LIN {X 272.582,Y -98.990,Z 143.292,A 160.041,B 90.000,C 0.000} C_DIS
LIN {X 272.604,Y -98.930,Z 143.343,A 160.054,B 90.000,C 0.000} C_DIS
LIN {X 272.618,Y -98.890,Z 143.394,A 160.062,B 90.000,C 0.000} C_DIS
LIN {X 272.688,Y -98.698,Z 143.436,A 160.103,B 90.000,C 0.000} C_DIS
LIN {X 272.717,Y -98.618,Z 143.538,A 160.119,B 90.000,C 0.000} C_DIS
LIN {X 272.786,Y -98.426,Z 143.581,A 160.160,B 90.000,C 0.000} C_DIS
LIN {X 272.801,Y -98.386,Z 143.632,A 160.168,B 90.000,C 0.000} C_DIS
LIN {X 272.822,Y -98.326,Z 143.683,A 160.181,B 90.000,C 0.000} C_DIS
LIN {X 272.926,Y -98.038,Z 143.725,A 160.241,B 90.000,C 0.000} C_DIS
LIN {X 272.947,Y -97.978,Z 143.776,A 160.254,B 90.000,C 0.000} C_DIS
LIN {X 272.962,Y -97.938,Z 143.827,A 160.262,B 90.000,C 0.000} C_DIS
LIN {X 273.031,Y -97.746,Z 143.870,A 160.302,B 90.000,C 0.000} C_DIS
LIN {X 273.059,Y -97.666,Z 143.972,A 160.319,B 90.000,C 0.000} C_DIS
LIN {X 273.128,Y -97.474,Z 144.014,A 160.360,B 90.000,C 0.000} C_DIS
LIN {X 273.142,Y -97.434,Z 144.065,A 160.368,B 90.000,C 0.000} C_DIS
LIN {X 273.164,Y -97.374,Z 144.116,A 160.380,B 90.000,C 0.000} C_DIS
LIN {X 273.266,Y -97.086,Z 144.159,A 160.441,B 90.000,C 0.000} C_DIS
LIN {X 273.287,Y -97.026,Z 144.210,A 160.454,B 90.000,C 0.000} C_DIS
LIN {X 273.302,Y -96.986,Z 144.261,A 160.462,B 90.000,C 0.000} C_DIS
LIN {X 273.370,Y -96.793,Z 144.303,A 160.502,B 90.000,C 0.000} C_DIS
LIN {X 273.398,Y -96.713,Z 144.405,A 160.519,B 90.000,C 0.000} C_DIS
LIN {X 273.466,Y -96.521,Z 144.448,A 160.559,B 90.000,C 0.000} C_DIS
LIN {X 273.480,Y -96.481,Z 144.499,A 160.568,B 90.000,C 0.000} C_DIS
LIN {X 273.502,Y -96.420,Z 144.550,A 160.580,B 90.000,C 0.000} C_DIS
LIN {X 273.603,Y -96.132,Z 144.592,A 160.641,B 90.000,C 0.000} C_DIS
LIN {X 273.624,Y -96.072,Z 144.644,A 160.653,B 90.000,C 0.000} C_DIS
LIN {X 273.638,Y -96.031,Z 144.695,A 160.662,B 90.000,C 0.000} C_DIS
LIN {X 273.706,Y -95.839,Z 144.737,A 160.702,B 90.000,C 0.000} C_DIS
LIN {X 273.734,Y -95.759,Z 144.839,A 160.719,B 90.000,C 0.000} C_DIS
LIN {X 273.801,Y -95.566,Z 144.882,A 160.759,B 90.000,C 0.000} C_DIS
LIN {X 273.815,Y -95.526,Z 144.933,A 160.768,B 90.000,C 0.000} C_DIS
LIN {X 273.836,Y -95.466,Z 144.984,A 160.780,B 90.000,C 0.000} C_DIS
LIN {X 273.937,Y -95.177,Z 145.026,A 160.841,B 90.000,C 0.000} C_DIS
LIN {X 273.958,Y -95.116,Z 145.077,A 160.853,B 90.000,C 0.000} C_DIS
LIN {X 273.972,Y -95.076,Z 145.128,A 160.862,B 90.000,C 0.000} C_DIS
LIN {X 274.039,Y -94.883,Z 145.171,A 160.902,B 90.000,C 0.000} C_DIS
LIN {X 274.066,Y -94.803,Z 145.273,A 160.919,B 90.000,C 0.000} C_DIS
LIN {X 274.133,Y -94.610,Z 145.315,A 160.959,B 90.000,C 0.000} C_DIS
LIN {X 274.161,Y -94.530,Z 145.417,A 160.976,B 90.000,C 0.000} C_DIS
LIN {X 274.227,Y -94.337,Z 145.460,A 161.016,B 90.000,C 0.000} C_DIS
LIN {X 274.241,Y -94.297,Z 145.511,A 161.025,B 90.000,C 0.000} C_DIS
LIN {X 274.262,Y -94.237,Z 145.562,A 161.037,B 90.000,C 0.000} C_DIS
LIN {X 274.361,Y -93.947,Z 145.604,A 161.098,B 90.000,C 0.000} C_DIS
LIN {X 274.382,Y -93.887,Z 145.655,A 161.110,B 90.000,C 0.000} C_DIS
LIN {X 274.395,Y -93.846,Z 145.706,A 161.119,B 90.000,C 0.000} C_DIS
LIN {X 274.461,Y -93.653,Z 145.749,A 161.159,B 90.000,C 0.000} C_DIS
LIN {X 274.475,Y -93.613,Z 145.800,A 161.167,B 90.000,C 0.000} C_DIS
LIN {X 274.496,Y -93.553,Z 145.851,A 161.180,B 90.000,C 0.000} C_DIS
LIN {X 274.594,Y -93.263,Z 145.893,A 161.241,B 90.000,C 0.000} C_DIS
LIN {X 274.615,Y -93.203,Z 145.944,A 161.253,B 90.000,C 0.000} C_DIS
LIN {X 274.628,Y -93.162,Z 145.995,A 161.261,B 90.000,C 0.000} C_DIS
LIN {X 274.694,Y -92.969,Z 146.038,A 161.302,B 90.000,C 0.000} C_DIS
LIN {X 274.721,Y -92.889,Z 146.140,A 161.319,B 90.000,C 0.000} C_DIS
LIN {X 274.786,Y -92.695,Z 146.182,A 161.359,B 90.000,C 0.000} C_DIS
LIN {X 274.814,Y -92.615,Z 146.284,A 161.376,B 90.000,C 0.000} C_DIS
LIN {X 274.879,Y -92.421,Z 146.327,A 161.416,B 90.000,C 0.000} C_DIS
LIN {X 274.892,Y -92.381,Z 146.378,A 161.424,B 90.000,C 0.000} C_DIS
LIN {X 274.913,Y -92.321,Z 146.429,A 161.437,B 90.000,C 0.000} C_DIS
LIN {X 275.010,Y -92.030,Z 146.471,A 161.498,B 90.000,C 0.000} C_DIS
LIN {X 275.030,Y -91.970,Z 146.522,A 161.510,B 90.000,C 0.000} C_DIS
LIN {X 275.044,Y -91.930,Z 146.573,A 161.518,B 90.000,C 0.000} C_DIS
LIN {X 275.108,Y -91.736,Z 146.616,A 161.559,B 90.000,C 0.000} C_DIS
LIN {X 275.135,Y -91.655,Z 146.718,A 161.576,B 90.000,C 0.000} C_DIS
LIN {X 275.199,Y -91.462,Z 146.760,A 161.616,B 90.000,C 0.000} C_DIS
LIN {X 275.213,Y -91.421,Z 146.811,A 161.624,B 90.000,C 0.000} C_DIS
LIN {X 275.233,Y -91.361,Z 146.862,A 161.637,B 90.000,C 0.000} C_DIS
LIN {X 275.329,Y -91.070,Z 146.905,A 161.697,B 90.000,C 0.000} C_DIS
LIN {X 275.349,Y -91.010,Z 146.956,A 161.710,B 90.000,C 0.000} C_DIS
LIN {X 275.363,Y -90.970,Z 147.007,A 161.718,B 90.000,C 0.000} C_DIS
LIN {X 275.427,Y -90.776,Z 147.049,A 161.759,B 90.000,C 0.000} C_DIS
LIN {X 275.453,Y -90.695,Z 147.152,A 161.775,B 90.000,C 0.000} C_DIS
LIN {X 275.517,Y -90.501,Z 147.194,A 161.816,B 90.000,C 0.000} C_DIS
LIN {X 275.530,Y -90.461,Z 147.245,A 161.824,B 90.000,C 0.000} C_DIS
LIN {X 275.550,Y -90.400,Z 147.296,A 161.837,B 90.000,C 0.000} C_DIS
LIN {X 275.645,Y -90.109,Z 147.338,A 161.897,B 90.000,C 0.000} C_DIS
LIN {X 275.665,Y -90.049,Z 147.390,A 161.910,B 90.000,C 0.000} C_DIS
LIN {X 275.678,Y -90.008,Z 147.441,A 161.918,B 90.000,C 0.000} C_DIS
LIN {X 275.742,Y -89.814,Z 147.483,A 161.959,B 90.000,C 0.000} C_DIS
LIN {X 275.768,Y -89.734,Z 147.585,A 161.975,B 90.000,C 0.000} C_DIS
LIN {X 275.831,Y -89.539,Z 147.628,A 162.016,B 90.000,C 0.000} C_DIS
LIN {X 275.844,Y -89.499,Z 147.679,A 162.024,B 90.000,C 0.000} C_DIS
LIN {X 275.864,Y -89.438,Z 147.730,A 162.037,B 90.000,C 0.000} C_DIS
LIN {X 275.958,Y -89.147,Z 147.772,A 162.097,B 90.000,C 0.000} C_DIS
LIN {X 275.978,Y -89.087,Z 147.823,A 162.110,B 90.000,C 0.000} C_DIS
LIN {X 275.991,Y -89.046,Z 147.874,A 162.118,B 90.000,C 0.000} C_DIS
LIN {X 276.053,Y -88.852,Z 147.917,A 162.158,B 90.000,C 0.000} C_DIS
LIN {X 276.079,Y -88.771,Z 148.019,A 162.175,B 90.000,C 0.000} C_DIS
LIN {X 276.142,Y -88.577,Z 148.061,A 162.216,B 90.000,C 0.000} C_DIS
LIN {X 276.155,Y -88.536,Z 148.112,A 162.224,B 90.000,C 0.000} C_DIS
LIN {X 276.174,Y -88.476,Z 148.163,A 162.237,B 90.000,C 0.000} C_DIS
LIN {X 276.267,Y -88.184,Z 148.206,A 162.297,B 90.000,C 0.000} C_DIS
LIN {X 276.287,Y -88.123,Z 148.257,A 162.310,B 90.000,C 0.000} C_DIS
LIN {X 276.300,Y -88.083,Z 148.308,A 162.318,B 90.000,C 0.000} C_DIS
LIN {X 276.361,Y -87.888,Z 148.350,A 162.358,B 90.000,C 0.000} C_DIS
LIN {X 276.387,Y -87.807,Z 148.452,A 162.375,B 90.000,C 0.000} C_DIS
LIN {X 276.449,Y -87.613,Z 148.495,A 162.415,B 90.000,C 0.000} C_DIS
LIN {X 276.462,Y -87.572,Z 148.546,A 162.424,B 90.000,C 0.000} C_DIS
LIN {X 276.481,Y -87.512,Z 148.597,A 162.436,B 90.000,C 0.000} C_DIS
LIN {X 276.573,Y -87.220,Z 148.639,A 162.497,B 90.000,C 0.000} C_DIS
LIN {X 276.592,Y -87.159,Z 148.690,A 162.510,B 90.000,C 0.000} C_DIS
LIN {X 276.605,Y -87.118,Z 148.741,A 162.518,B 90.000,C 0.000} C_DIS
LIN {X 276.666,Y -86.924,Z 148.784,A 162.558,B 90.000,C 0.000} C_DIS
LIN {X 276.692,Y -86.843,Z 148.886,A 162.575,B 90.000,C 0.000} C_DIS
LIN {X 276.753,Y -86.648,Z 148.928,A 162.615,B 90.000,C 0.000} C_DIS
LIN {X 276.766,Y -86.607,Z 148.979,A 162.624,B 90.000,C 0.000} C_DIS
LIN {X 276.785,Y -86.546,Z 149.030,A 162.636,B 90.000,C 0.000} C_DIS
LIN {X 276.876,Y -86.254,Z 149.073,A 162.697,B 90.000,C 0.000} C_DIS
LIN {X 276.895,Y -86.193,Z 149.124,A 162.709,B 90.000,C 0.000} C_DIS
LIN {X 276.907,Y -86.153,Z 149.175,A 162.718,B 90.000,C 0.000} C_DIS
LIN {X 276.968,Y -85.958,Z 149.217,A 162.758,B 90.000,C 0.000} C_DIS
LIN {X 276.993,Y -85.877,Z 149.319,A 162.775,B 90.000,C 0.000} C_DIS
LIN {X 277.053,Y -85.682,Z 149.362,A 162.815,B 90.000,C 0.000} C_DIS
LIN {X 277.066,Y -85.641,Z 149.413,A 162.824,B 90.000,C 0.000} C_DIS
LIN {X 277.085,Y -85.580,Z 149.464,A 162.836,B 90.000,C 0.000} C_DIS
LIN {X 277.175,Y -85.288,Z 149.506,A 162.897,B 90.000,C 0.000} C_DIS
LIN {X 277.194,Y -85.227,Z 149.557,A 162.909,B 90.000,C 0.000} C_DIS
LIN {X 277.206,Y -85.186,Z 149.608,A 162.918,B 90.000,C 0.000} C_DIS
LIN {X 277.266,Y -84.991,Z 149.651,A 162.958,B 90.000,C 0.000} C_DIS
LIN {X 277.291,Y -84.910,Z 149.753,A 162.975,B 90.000,C 0.000} C_DIS
LIN {X 277.351,Y -84.715,Z 149.795,A 163.015,B 90.000,C 0.000} C_DIS
LIN {X 277.363,Y -84.674,Z 149.847,A 163.023,B 90.000,C 0.000} C_DIS
LIN {X 277.382,Y -84.613,Z 149.898,A 163.036,B 90.000,C 0.000} C_DIS
LIN {X 277.471,Y -84.320,Z 149.940,A 163.097,B 90.000,C 0.000} C_DIS
LIN {X 277.489,Y -84.259,Z 149.991,A 163.109,B 90.000,C 0.000} C_DIS
LIN {X 277.502,Y -84.219,Z 150.042,A 163.118,B 90.000,C 0.000} C_DIS
LIN {X 277.561,Y -84.023,Z 150.085,A 163.158,B 90.000,C 0.000} C_DIS
LIN {X 277.586,Y -83.942,Z 150.187,A 163.175,B 90.000,C 0.000} C_DIS
LIN {X 277.645,Y -83.747,Z 150.229,A 163.215,B 90.000,C 0.000} C_DIS
LIN {X 277.657,Y -83.706,Z 150.280,A 163.223,B 90.000,C 0.000} C_DIS
LIN {X 277.675,Y -83.645,Z 150.331,A 163.236,B 90.000,C 0.000} C_DIS
LIN {X 277.763,Y -83.352,Z 150.374,A 163.296,B 90.000,C 0.000} C_DIS
LIN {X 277.782,Y -83.291,Z 150.425,A 163.309,B 90.000,C 0.000} C_DIS
LIN {X 277.794,Y -83.250,Z 150.476,A 163.317,B 90.000,C 0.000} C_DIS
LIN {X 277.852,Y -83.055,Z 150.518,A 163.358,B 90.000,C 0.000} C_DIS
LIN {X 277.877,Y -82.973,Z 150.620,A 163.375,B 90.000,C 0.000} C_DIS
LIN {X 277.935,Y -82.778,Z 150.663,A 163.415,B 90.000,C 0.000} C_DIS
LIN {X 277.947,Y -82.737,Z 150.714,A 163.423,B 90.000,C 0.000} C_DIS
LIN {X 277.965,Y -82.676,Z 150.765,A 163.436,B 90.000,C 0.000} C_DIS
LIN {X 278.052,Y -82.382,Z 150.807,A 163.496,B 90.000,C 0.000} C_DIS
LIN {X 278.071,Y -82.321,Z 150.858,A 163.509,B 90.000,C 0.000} C_DIS
LIN {X 278.083,Y -82.280,Z 150.909,A 163.517,B 90.000,C 0.000} C_DIS
LIN {X 278.140,Y -82.085,Z 150.952,A 163.558,B 90.000,C 0.000} C_DIS
LIN {X 278.164,Y -82.003,Z 151.054,A 163.574,B 90.000,C 0.000} C_DIS
LIN {X 278.222,Y -81.807,Z 151.096,A 163.615,B 90.000,C 0.000} C_DIS
LIN {X 278.234,Y -81.767,Z 151.147,A 163.623,B 90.000,C 0.000} C_DIS
LIN {X 278.252,Y -81.706,Z 151.198,A 163.636,B 90.000,C 0.000} C_DIS
LIN {X 278.338,Y -81.412,Z 151.241,A 163.696,B 90.000,C 0.000} C_DIS
LIN {X 278.356,Y -81.351,Z 151.292,A 163.709,B 90.000,C 0.000} C_DIS
LIN {X 278.368,Y -81.310,Z 151.343,A 163.717,B 90.000,C 0.000} C_DIS
LIN {X 278.425,Y -81.114,Z 151.385,A 163.758,B 90.000,C 0.000} C_DIS
LIN {X 278.449,Y -81.032,Z 151.487,A 163.774,B 90.000,C 0.000} C_DIS
LIN {X 278.506,Y -80.836,Z 151.530,A 163.815,B 90.000,C 0.000} C_DIS
LIN {X 278.518,Y -80.796,Z 151.581,A 163.823,B 90.000,C 0.000} C_DIS
LIN {X 278.535,Y -80.734,Z 151.632,A 163.836,B 90.000,C 0.000} C_DIS
LIN {X 278.620,Y -80.440,Z 151.674,A 163.896,B 90.000,C 0.000} C_DIS
LIN {X 278.638,Y -80.379,Z 151.725,A 163.909,B 90.000,C 0.000} C_DIS
LIN {X 278.650,Y -80.338,Z 151.776,A 163.917,B 90.000,C 0.000} C_DIS
LIN {X 278.706,Y -80.142,Z 151.819,A 163.957,B 90.000,C 0.000} C_DIS
LIN {X 278.730,Y -80.060,Z 151.921,A 163.974,B 90.000,C 0.000} C_DIS
LIN {X 278.786,Y -79.864,Z 151.963,A 164.015,B 90.000,C 0.000} C_DIS
LIN {X 278.798,Y -79.823,Z 152.014,A 164.023,B 90.000,C 0.000} C_DIS
LIN {X 278.815,Y -79.762,Z 152.065,A 164.035,B 90.000,C 0.000} C_DIS
LIN {X 278.899,Y -79.468,Z 152.108,A 164.096,B 90.000,C 0.000} C_DIS
LIN {X 278.917,Y -79.406,Z 152.159,A 164.109,B 90.000,C 0.000} C_DIS
LIN {X 278.928,Y -79.366,Z 152.210,A 164.117,B 90.000,C 0.000} C_DIS
LIN {X 278.984,Y -79.169,Z 152.252,A 164.157,B 90.000,C 0.000} C_DIS
LIN {X 279.007,Y -79.088,Z 152.355,A 164.174,B 90.000,C 0.000} C_DIS
LIN {X 279.063,Y -78.891,Z 152.397,A 164.214,B 90.000,C 0.000} C_DIS
LIN {X 279.075,Y -78.850,Z 152.448,A 164.223,B 90.000,C 0.000} C_DIS
LIN {X 279.092,Y -78.789,Z 152.499,A 164.235,B 90.000,C 0.000} C_DIS
LIN {X 279.175,Y -78.494,Z 152.542,A 164.296,B 90.000,C 0.000} C_DIS
LIN {X 279.192,Y -78.433,Z 152.593,A 164.308,B 90.000,C 0.000} C_DIS
LIN {X 279.204,Y -78.392,Z 152.644,A 164.317,B 90.000,C 0.000} C_DIS
LIN {X 279.259,Y -78.196,Z 152.686,A 164.357,B 90.000,C 0.000} C_DIS
LIN {X 279.282,Y -78.114,Z 152.788,A 164.374,B 90.000,C 0.000} C_DIS
LIN {X 279.337,Y -77.917,Z 152.831,A 164.414,B 90.000,C 0.000} C_DIS
LIN {X 279.348,Y -77.876,Z 152.882,A 164.423,B 90.000,C 0.000} C_DIS
LIN {X 279.365,Y -77.815,Z 152.933,A 164.435,B 90.000,C 0.000} C_DIS
LIN {X 279.447,Y -77.520,Z 152.975,A 164.496,B 90.000,C 0.000} C_DIS
LIN {X 279.464,Y -77.459,Z 153.026,A 164.508,B 90.000,C 0.000} C_DIS
LIN {X 279.475,Y -77.418,Z 153.077,A 164.517,B 90.000,C 0.000} C_DIS
LIN {X 279.530,Y -77.221,Z 153.120,A 164.557,B 90.000,C 0.000} C_DIS
LIN {X 279.552,Y -77.139,Z 153.222,A 164.574,B 90.000,C 0.000} C_DIS
LIN {X 279.607,Y -76.942,Z 153.264,A 164.614,B 90.000,C 0.000} C_DIS
LIN {X 279.618,Y -76.901,Z 153.315,A 164.623,B 90.000,C 0.000} C_DIS
LIN {X 279.635,Y -76.840,Z 153.366,A 164.635,B 90.000,C 0.000} C_DIS
LIN {X 279.716,Y -76.545,Z 153.409,A 164.696,B 90.000,C 0.000} C_DIS
LIN {X 279.733,Y -76.483,Z 153.460,A 164.708,B 90.000,C 0.000} C_DIS
LIN {X 279.744,Y -76.442,Z 153.511,A 164.717,B 90.000,C 0.000} C_DIS
LIN {X 279.798,Y -76.245,Z 153.553,A 164.757,B 90.000,C 0.000} C_DIS
LIN {X 279.820,Y -76.163,Z 153.655,A 164.774,B 90.000,C 0.000} C_DIS
LIN {X 279.873,Y -75.966,Z 153.698,A 164.814,B 90.000,C 0.000} C_DIS
LIN {X 279.896,Y -75.884,Z 153.800,A 164.831,B 90.000,C 0.000} C_DIS
LIN {X 279.949,Y -75.687,Z 153.842,A 164.871,B 90.000,C 0.000} C_DIS
LIN {X 279.960,Y -75.646,Z 153.893,A 164.880,B 90.000,C 0.000} C_DIS
LIN {X 279.977,Y -75.585,Z 153.944,A 164.892,B 90.000,C 0.000} C_DIS
LIN {X 280.056,Y -75.289,Z 153.987,A 164.953,B 90.000,C 0.000} C_DIS
LIN {X 280.073,Y -75.228,Z 154.038,A 164.965,B 90.000,C 0.000} C_DIS
LIN {X 280.084,Y -75.187,Z 154.089,A 164.974,B 90.000,C 0.000} C_DIS
LIN {X 280.137,Y -74.989,Z 154.131,A 165.014,B 90.000,C 0.000} C_DIS
LIN {X 280.148,Y -74.948,Z 154.182,A 165.022,B 90.000,C 0.000} C_DIS
LIN {X 280.164,Y -74.887,Z 154.233,A 165.035,B 90.000,C 0.000} C_DIS
LIN {X 280.243,Y -74.591,Z 154.276,A 165.095,B 90.000,C 0.000} C_DIS
LIN {X 280.259,Y -74.529,Z 154.327,A 165.108,B 90.000,C 0.000} C_DIS
LIN {X 280.270,Y -74.488,Z 154.378,A 165.116,B 90.000,C 0.000} C_DIS
LIN {X 280.323,Y -74.291,Z 154.420,A 165.157,B 90.000,C 0.000} C_DIS
LIN {X 280.344,Y -74.209,Z 154.522,A 165.173,B 90.000,C 0.000} C_DIS
LIN {X 280.397,Y -74.012,Z 154.565,A 165.214,B 90.000,C 0.000} C_DIS
LIN {X 280.418,Y -73.930,Z 154.667,A 165.231,B 90.000,C 0.000} C_DIS
LIN {X 280.470,Y -73.732,Z 154.709,A 165.271,B 90.000,C 0.000} C_DIS
LIN {X 280.481,Y -73.691,Z 154.760,A 165.279,B 90.000,C 0.000} C_DIS
LIN {X 280.497,Y -73.630,Z 154.812,A 165.292,B 90.000,C 0.000} C_DIS
LIN {X 280.575,Y -73.333,Z 154.854,A 165.352,B 90.000,C 0.000} C_DIS
LIN {X 280.591,Y -73.272,Z 154.905,A 165.365,B 90.000,C 0.000} C_DIS
LIN {X 280.602,Y -73.231,Z 154.956,A 165.373,B 90.000,C 0.000} C_DIS
LIN {X 280.653,Y -73.033,Z 154.998,A 165.414,B 90.000,C 0.000} C_DIS
LIN {X 280.674,Y -72.951,Z 155.101,A 165.430,B 90.000,C 0.000} C_DIS
LIN {X 280.726,Y -72.753,Z 155.143,A 165.471,B 90.000,C 0.000} C_DIS
LIN {X 280.736,Y -72.712,Z 155.194,A 165.479,B 90.000,C 0.000} C_DIS
LIN {X 280.752,Y -72.651,Z 155.245,A 165.492,B 90.000,C 0.000} C_DIS
LIN {X 280.829,Y -72.354,Z 155.288,A 165.552,B 90.000,C 0.000} C_DIS
LIN {X 280.845,Y -72.292,Z 155.339,A 165.565,B 90.000,C 0.000} C_DIS
LIN {X 280.855,Y -72.251,Z 155.390,A 165.573,B 90.000,C 0.000} C_DIS
LIN {X 280.906,Y -72.054,Z 155.432,A 165.614,B 90.000,C 0.000} C_DIS
LIN {X 280.927,Y -71.971,Z 155.534,A 165.630,B 90.000,C 0.000} C_DIS
LIN {X 280.978,Y -71.773,Z 155.577,A 165.671,B 90.000,C 0.000} C_DIS
LIN {X 280.988,Y -71.732,Z 155.628,A 165.679,B 90.000,C 0.000} C_DIS
LIN {X 281.004,Y -71.671,Z 155.679,A 165.692,B 90.000,C 0.000} C_DIS
LIN {X 281.080,Y -71.374,Z 155.721,A 165.752,B 90.000,C 0.000} C_DIS
LIN {X 281.095,Y -71.312,Z 155.772,A 165.765,B 90.000,C 0.000} C_DIS
LIN {X 281.106,Y -71.271,Z 155.823,A 165.773,B 90.000,C 0.000} C_DIS
LIN {X 281.156,Y -71.073,Z 155.866,A 165.813,B 90.000,C 0.000} C_DIS
LIN {X 281.177,Y -70.991,Z 155.968,A 165.830,B 90.000,C 0.000} C_DIS
LIN {X 281.227,Y -70.793,Z 156.010,A 165.871,B 90.000,C 0.000} C_DIS
LIN {X 281.237,Y -70.752,Z 156.061,A 165.879,B 90.000,C 0.000} C_DIS
LIN {X 281.252,Y -70.690,Z 156.112,A 165.892,B 90.000,C 0.000} C_DIS
LIN {X 281.327,Y -70.393,Z 156.155,A 165.952,B 90.000,C 0.000} C_DIS
LIN {X 281.342,Y -70.331,Z 156.206,A 165.965,B 90.000,C 0.000} C_DIS
LIN {X 281.353,Y -70.290,Z 156.257,A 165.973,B 90.000,C 0.000} C_DIS
LIN {X 281.402,Y -70.092,Z 156.299,A 166.013,B 90.000,C 0.000} C_DIS
LIN {X 281.423,Y -70.009,Z 156.401,A 166.030,B 90.000,C 0.000} C_DIS
LIN {X 281.472,Y -69.811,Z 156.444,A 166.070,B 90.000,C 0.000} C_DIS
LIN {X 281.482,Y -69.770,Z 156.495,A 166.079,B 90.000,C 0.000} C_DIS
LIN {X 281.497,Y -69.708,Z 156.546,A 166.091,B 90.000,C 0.000} C_DIS
LIN {X 281.571,Y -69.411,Z 156.588,A 166.152,B 90.000,C 0.000} C_DIS
LIN {X 281.586,Y -69.349,Z 156.639,A 166.165,B 90.000,C 0.000} C_DIS
LIN {X 281.596,Y -69.308,Z 156.690,A 166.173,B 90.000,C 0.000} C_DIS
LIN {X 281.645,Y -69.110,Z 156.733,A 166.213,B 90.000,C 0.000} C_DIS
LIN {X 281.665,Y -69.027,Z 156.835,A 166.230,B 90.000,C 0.000} C_DIS
LIN {X 281.714,Y -68.829,Z 156.877,A 166.270,B 90.000,C 0.000} C_DIS
LIN {X 281.724,Y -68.788,Z 156.928,A 166.279,B 90.000,C 0.000} C_DIS
LIN {X 281.739,Y -68.726,Z 156.979,A 166.291,B 90.000,C 0.000} C_DIS
LIN {X 281.811,Y -68.428,Z 157.022,A 166.352,B 90.000,C 0.000} C_DIS
LIN {X 281.826,Y -68.366,Z 157.073,A 166.364,B 90.000,C 0.000} C_DIS
LIN {X 281.836,Y -68.325,Z 157.124,A 166.373,B 90.000,C 0.000} C_DIS
LIN {X 281.884,Y -68.127,Z 157.166,A 166.413,B 90.000,C 0.000} C_DIS
LIN {X 281.904,Y -68.044,Z 157.268,A 166.430,B 90.000,C 0.000} C_DIS
LIN {X 281.952,Y -67.846,Z 157.311,A 166.470,B 90.000,C 0.000} C_DIS
LIN {X 281.962,Y -67.804,Z 157.362,A 166.479,B 90.000,C 0.000} C_DIS
LIN {X 281.977,Y -67.743,Z 157.413,A 166.491,B 90.000,C 0.000} C_DIS
LIN {X 282.048,Y -67.445,Z 157.455,A 166.552,B 90.000,C 0.000} C_DIS
LIN {X 282.063,Y -67.383,Z 157.506,A 166.564,B 90.000,C 0.000} C_DIS
LIN {X 282.073,Y -67.342,Z 157.558,A 166.573,B 90.000,C 0.000} C_DIS
LIN {X 282.120,Y -67.143,Z 157.600,A 166.613,B 90.000,C 0.000} C_DIS
LIN {X 282.140,Y -67.060,Z 157.702,A 166.630,B 90.000,C 0.000} C_DIS
LIN {X 282.187,Y -66.862,Z 157.745,A 166.670,B 90.000,C 0.000} C_DIS
LIN {X 282.197,Y -66.820,Z 157.796,A 166.678,B 90.000,C 0.000} C_DIS
LIN {X 282.211,Y -66.758,Z 157.847,A 166.691,B 90.000,C 0.000} C_DIS
LIN {X 282.282,Y -66.460,Z 157.889,A 166.752,B 90.000,C 0.000} C_DIS
LIN {X 282.296,Y -66.398,Z 157.940,A 166.764,B 90.000,C 0.000} C_DIS
LIN {X 282.306,Y -66.357,Z 157.991,A 166.773,B 90.000,C 0.000} C_DIS
LIN {X 282.353,Y -66.158,Z 158.034,A 166.813,B 90.000,C 0.000} C_DIS
LIN {X 282.372,Y -66.076,Z 158.136,A 166.830,B 90.000,C 0.000} C_DIS
LIN {X 282.419,Y -65.877,Z 158.178,A 166.870,B 90.000,C 0.000} C_DIS
LIN {X 282.428,Y -65.836,Z 158.229,A 166.878,B 90.000,C 0.000} C_DIS
LIN {X 282.443,Y -65.773,Z 158.280,A 166.891,B 90.000,C 0.000} C_DIS
LIN {X 282.512,Y -65.475,Z 158.323,A 166.951,B 90.000,C 0.000} C_DIS
LIN {X 282.526,Y -65.413,Z 158.374,A 166.964,B 90.000,C 0.000} C_DIS
LIN {X 282.536,Y -65.372,Z 158.425,A 166.972,B 90.000,C 0.000} C_DIS
LIN {X 282.582,Y -65.173,Z 158.467,A 167.013,B 90.000,C 0.000} C_DIS
LIN {X 282.601,Y -65.090,Z 158.569,A 167.030,B 90.000,C 0.000} C_DIS
LIN {X 282.647,Y -64.891,Z 158.612,A 167.070,B 90.000,C 0.000} C_DIS
LIN {X 282.656,Y -64.850,Z 158.663,A 167.078,B 90.000,C 0.000} C_DIS
LIN {X 282.670,Y -64.788,Z 158.714,A 167.091,B 90.000,C 0.000} C_DIS
LIN {X 282.739,Y -64.489,Z 158.756,A 167.151,B 90.000,C 0.000} C_DIS
LIN {X 282.753,Y -64.427,Z 158.807,A 167.164,B 90.000,C 0.000} C_DIS
LIN {X 282.762,Y -64.386,Z 158.858,A 167.172,B 90.000,C 0.000} C_DIS
LIN {X 282.807,Y -64.187,Z 158.901,A 167.213,B 90.000,C 0.000} C_DIS
LIN {X 282.826,Y -64.104,Z 159.003,A 167.229,B 90.000,C 0.000} C_DIS
LIN {X 282.871,Y -63.905,Z 159.045,A 167.270,B 90.000,C 0.000} C_DIS
LIN {X 282.881,Y -63.863,Z 159.096,A 167.278,B 90.000,C 0.000} C_DIS
LIN {X 282.895,Y -63.801,Z 159.147,A 167.291,B 90.000,C 0.000} C_DIS
LIN {X 282.962,Y -63.502,Z 159.190,A 167.351,B 90.000,C 0.000} C_DIS
LIN {X 282.976,Y -63.440,Z 159.241,A 167.364,B 90.000,C 0.000} C_DIS
LIN {X 282.985,Y -63.399,Z 159.292,A 167.372,B 90.000,C 0.000} C_DIS
LIN {X 283.030,Y -63.200,Z 159.334,A 167.413,B 90.000,C 0.000} C_DIS
LIN {X 283.048,Y -63.117,Z 159.436,A 167.429,B 90.000,C 0.000} C_DIS
LIN {X 283.093,Y -62.918,Z 159.479,A 167.470,B 90.000,C 0.000} C_DIS
LIN {X 283.102,Y -62.876,Z 159.530,A 167.478,B 90.000,C 0.000} C_DIS
LIN {X 283.116,Y -62.814,Z 159.581,A 167.491,B 90.000,C 0.000} C_DIS
LIN {X 283.182,Y -62.515,Z 159.623,A 167.551,B 90.000,C 0.000} C_DIS
LIN {X 283.195,Y -62.453,Z 159.674,A 167.564,B 90.000,C 0.000} C_DIS
LIN {X 283.205,Y -62.411,Z 159.725,A 167.572,B 90.000,C 0.000} C_DIS
LIN {X 283.248,Y -62.212,Z 159.768,A 167.612,B 90.000,C 0.000} C_DIS
LIN {X 283.267,Y -62.129,Z 159.870,A 167.629,B 90.000,C 0.000} C_DIS
LIN {X 283.310,Y -61.930,Z 159.912,A 167.670,B 90.000,C 0.000} C_DIS
LIN {X 283.319,Y -61.888,Z 159.963,A 167.678,B 90.000,C 0.000} C_DIS
LIN {X 283.333,Y -61.826,Z 160.015,A 167.690,B 90.000,C 0.000} C_DIS
LIN {X 283.398,Y -61.527,Z 160.057,A 167.751,B 90.000,C 0.000} C_DIS
LIN {X 283.412,Y -61.464,Z 160.108,A 167.764,B 90.000,C 0.000} C_DIS
LIN {X 283.421,Y -61.423,Z 160.159,A 167.772,B 90.000,C 0.000} C_DIS
LIN {X 283.464,Y -61.223,Z 160.201,A 167.812,B 90.000,C 0.000} C_DIS
LIN {X 283.482,Y -61.140,Z 160.304,A 167.829,B 90.000,C 0.000} C_DIS
LIN {X 283.525,Y -60.941,Z 160.346,A 167.869,B 90.000,C 0.000} C_DIS
LIN {X 283.534,Y -60.899,Z 160.397,A 167.878,B 90.000,C 0.000} C_DIS
LIN {X 283.547,Y -60.837,Z 160.448,A 167.890,B 90.000,C 0.000} C_DIS
LIN {X 283.611,Y -60.538,Z 160.491,A 167.951,B 90.000,C 0.000} C_DIS
LIN {X 283.624,Y -60.475,Z 160.542,A 167.963,B 90.000,C 0.000} C_DIS
LIN {X 283.633,Y -60.434,Z 160.593,A 167.972,B 90.000,C 0.000} C_DIS
LIN {X 283.676,Y -60.234,Z 160.635,A 168.012,B 90.000,C 0.000} C_DIS
LIN {X 283.693,Y -60.151,Z 160.737,A 168.029,B 90.000,C 0.000} C_DIS
LIN {X 283.736,Y -59.951,Z 160.780,A 168.069,B 90.000,C 0.000} C_DIS
LIN {X 283.744,Y -59.910,Z 160.831,A 168.078,B 90.000,C 0.000} C_DIS
LIN {X 283.757,Y -59.848,Z 160.882,A 168.090,B 90.000,C 0.000} C_DIS
LIN {X 283.820,Y -59.548,Z 160.924,A 168.151,B 90.000,C 0.000} C_DIS
LIN {X 283.834,Y -59.486,Z 160.975,A 168.163,B 90.000,C 0.000} C_DIS
LIN {X 283.842,Y -59.444,Z 161.026,A 168.172,B 90.000,C 0.000} C_DIS
LIN {X 283.884,Y -59.244,Z 161.069,A 168.212,B 90.000,C 0.000} C_DIS
LIN {X 283.901,Y -59.161,Z 161.171,A 168.229,B 90.000,C 0.000} C_DIS
LIN {X 283.943,Y -58.961,Z 161.213,A 168.269,B 90.000,C 0.000} C_DIS
LIN {X 283.952,Y -58.920,Z 161.264,A 168.278,B 90.000,C 0.000} C_DIS
LIN {X 283.964,Y -58.857,Z 161.315,A 168.290,B 90.000,C 0.000} C_DIS
LIN {X 284.026,Y -58.557,Z 161.358,A 168.351,B 90.000,C 0.000} C_DIS
LIN {X 284.039,Y -58.495,Z 161.409,A 168.363,B 90.000,C 0.000} C_DIS
LIN {X 284.048,Y -58.453,Z 161.460,A 168.372,B 90.000,C 0.000} C_DIS
LIN {X 284.089,Y -58.253,Z 161.502,A 168.412,B 90.000,C 0.000} C_DIS
LIN {X 284.106,Y -58.170,Z 161.604,A 168.429,B 90.000,C 0.000} C_DIS
LIN {X 284.147,Y -57.970,Z 161.647,A 168.469,B 90.000,C 0.000} C_DIS
LIN {X 284.155,Y -57.929,Z 161.698,A 168.477,B 90.000,C 0.000} C_DIS
LIN {X 284.168,Y -57.866,Z 161.749,A 168.490,B 90.000,C 0.000} C_DIS
LIN {X 284.229,Y -57.566,Z 161.791,A 168.551,B 90.000,C 0.000} C_DIS
LIN {X 284.242,Y -57.504,Z 161.842,A 168.563,B 90.000,C 0.000} C_DIS
LIN {X 284.250,Y -57.462,Z 161.893,A 168.571,B 90.000,C 0.000} C_DIS
LIN {X 284.290,Y -57.262,Z 161.936,A 168.612,B 90.000,C 0.000} C_DIS
LIN {X 284.307,Y -57.179,Z 162.038,A 168.629,B 90.000,C 0.000} C_DIS
LIN {X 284.347,Y -56.979,Z 162.080,A 168.669,B 90.000,C 0.000} C_DIS
LIN {X 284.356,Y -56.937,Z 162.131,A 168.677,B 90.000,C 0.000} C_DIS
LIN {X 284.368,Y -56.875,Z 162.182,A 168.690,B 90.000,C 0.000} C_DIS
LIN {X 284.428,Y -56.574,Z 162.225,A 168.750,B 90.000,C 0.000} C_DIS
LIN {X 284.441,Y -56.512,Z 162.276,A 168.763,B 90.000,C 0.000} C_DIS
LIN {X 284.449,Y -56.470,Z 162.327,A 168.771,B 90.000,C 0.000} C_DIS
LIN {X 284.488,Y -56.270,Z 162.369,A 168.812,B 90.000,C 0.000} C_DIS
LIN {X 284.505,Y -56.187,Z 162.471,A 168.828,B 90.000,C 0.000} C_DIS
LIN {X 284.544,Y -55.986,Z 162.514,A 168.869,B 90.000,C 0.000} C_DIS
LIN {X 284.553,Y -55.945,Z 162.565,A 168.877,B 90.000,C 0.000} C_DIS
LIN {X 284.565,Y -55.882,Z 162.616,A 168.890,B 90.000,C 0.000} C_DIS
LIN {X 284.624,Y -55.582,Z 162.658,A 168.950,B 90.000,C 0.000} C_DIS
LIN {X 284.636,Y -55.519,Z 162.710,A 168.963,B 90.000,C 0.000} C_DIS
LIN {X 284.644,Y -55.477,Z 162.761,A 168.971,B 90.000,C 0.000} C_DIS
LIN {X 284.683,Y -55.277,Z 162.803,A 169.012,B 90.000,C 0.000} C_DIS
LIN {X 284.699,Y -55.194,Z 162.905,A 169.028,B 90.000,C 0.000} C_DIS
LIN {X 284.738,Y -54.993,Z 162.948,A 169.069,B 90.000,C 0.000} C_DIS
LIN {X 284.746,Y -54.952,Z 162.999,A 169.077,B 90.000,C 0.000} C_DIS
LIN {X 284.758,Y -54.889,Z 163.050,A 169.090,B 90.000,C 0.000} C_DIS
LIN {X 284.816,Y -54.588,Z 163.092,A 169.150,B 90.000,C 0.000} C_DIS
LIN {X 284.828,Y -54.526,Z 163.143,A 169.163,B 90.000,C 0.000} C_DIS
LIN {X 284.836,Y -54.484,Z 163.194,A 169.171,B 90.000,C 0.000} C_DIS
LIN {X 284.874,Y -54.284,Z 163.237,A 169.211,B 90.000,C 0.000} C_DIS
LIN {X 284.890,Y -54.200,Z 163.339,A 169.228,B 90.000,C 0.000} C_DIS
LIN {X 284.928,Y -54.000,Z 163.381,A 169.269,B 90.000,C 0.000} C_DIS
LIN {X 284.936,Y -53.958,Z 163.432,A 169.277,B 90.000,C 0.000} C_DIS
LIN {X 284.948,Y -53.895,Z 163.483,A 169.290,B 90.000,C 0.000} C_DIS
LIN {X 285.005,Y -53.594,Z 163.526,A 169.350,B 90.000,C 0.000} C_DIS
LIN {X 285.016,Y -53.532,Z 163.577,A 169.363,B 90.000,C 0.000} C_DIS
LIN {X 285.024,Y -53.490,Z 163.628,A 169.371,B 90.000,C 0.000} C_DIS
LIN {X 285.062,Y -53.289,Z 163.670,A 169.411,B 90.000,C 0.000} C_DIS
LIN {X 285.077,Y -53.206,Z 163.772,A 169.428,B 90.000,C 0.000} C_DIS
LIN {X 285.115,Y -53.005,Z 163.815,A 169.468,B 90.000,C 0.000} C_DIS
LIN {X 285.130,Y -52.922,Z 163.917,A 169.485,B 90.000,C 0.000} C_DIS
LIN {X 285.167,Y -52.721,Z 163.959,A 169.526,B 90.000,C 0.000} C_DIS
LIN {X 285.175,Y -52.679,Z 164.010,A 169.534,B 90.000,C 0.000} C_DIS
LIN {X 285.187,Y -52.617,Z 164.061,A 169.547,B 90.000,C 0.000} C_DIS
LIN {X 285.242,Y -52.316,Z 164.104,A 169.607,B 90.000,C 0.000} C_DIS
LIN {X 285.254,Y -52.253,Z 164.155,A 169.620,B 90.000,C 0.000} C_DIS
LIN {X 285.261,Y -52.211,Z 164.206,A 169.628,B 90.000,C 0.000} C_DIS
LIN {X 285.298,Y -52.010,Z 164.248,A 169.668,B 90.000,C 0.000} C_DIS
LIN {X 285.313,Y -51.927,Z 164.350,A 169.685,B 90.000,C 0.000} C_DIS
LIN {X 285.350,Y -51.726,Z 164.393,A 169.725,B 90.000,C 0.000} C_DIS
LIN {X 285.357,Y -51.684,Z 164.444,A 169.734,B 90.000,C 0.000} C_DIS
LIN {X 285.369,Y -51.621,Z 164.495,A 169.746,B 90.000,C 0.000} C_DIS
LIN {X 285.423,Y -51.320,Z 164.537,A 169.807,B 90.000,C 0.000} C_DIS
LIN {X 285.434,Y -51.257,Z 164.588,A 169.820,B 90.000,C 0.000} C_DIS
LIN {X 285.442,Y -51.216,Z 164.639,A 169.828,B 90.000,C 0.000} C_DIS
LIN {X 285.478,Y -51.015,Z 164.682,A 169.868,B 90.000,C 0.000} C_DIS
LIN {X 285.493,Y -50.931,Z 164.784,A 169.885,B 90.000,C 0.000} C_DIS
LIN {X 285.528,Y -50.730,Z 164.826,A 169.925,B 90.000,C 0.000} C_DIS
LIN {X 285.536,Y -50.688,Z 164.877,A 169.934,B 90.000,C 0.000} C_DIS
LIN {X 285.547,Y -50.626,Z 164.928,A 169.946,B 90.000,C 0.000} C_DIS
LIN {X 285.600,Y -50.324,Z 164.971,A 170.007,B 90.000,C 0.000} C_DIS
LIN {X 285.611,Y -50.261,Z 165.022,A 170.019,B 90.000,C 0.000} C_DIS
LIN {X 285.619,Y -50.220,Z 165.073,A 170.028,B 90.000,C 0.000} C_DIS
LIN {X 285.654,Y -50.018,Z 165.115,A 170.068,B 90.000,C 0.000} C_DIS
LIN {X 285.669,Y -49.935,Z 165.218,A 170.085,B 90.000,C 0.000} C_DIS
LIN {X 285.704,Y -49.734,Z 165.260,A 170.125,B 90.000,C 0.000} C_DIS
LIN {X 285.711,Y -49.692,Z 165.311,A 170.134,B 90.000,C 0.000} C_DIS
LIN {X 285.722,Y -49.629,Z 165.362,A 170.146,B 90.000,C 0.000} C_DIS
LIN {X 285.774,Y -49.327,Z 165.405,A 170.207,B 90.000,C 0.000} C_DIS
LIN {X 285.785,Y -49.265,Z 165.456,A 170.219,B 90.000,C 0.000} C_DIS
LIN {X 285.792,Y -49.223,Z 165.507,A 170.228,B 90.000,C 0.000} C_DIS
LIN {X 285.827,Y -49.022,Z 165.549,A 170.268,B 90.000,C 0.000} C_DIS
LIN {X 285.841,Y -48.938,Z 165.651,A 170.285,B 90.000,C 0.000} C_DIS
LIN {X 285.875,Y -48.737,Z 165.694,A 170.325,B 90.000,C 0.000} C_DIS
LIN {X 285.883,Y -48.695,Z 165.745,A 170.333,B 90.000,C 0.000} C_DIS
LIN {X 285.893,Y -48.632,Z 165.796,A 170.346,B 90.000,C 0.000} C_DIS
LIN {X 285.944,Y -48.330,Z 165.838,A 170.407,B 90.000,C 0.000} C_DIS
LIN {X 285.955,Y -48.267,Z 165.889,A 170.419,B 90.000,C 0.000} C_DIS
LIN {X 285.962,Y -48.225,Z 165.940,A 170.428,B 90.000,C 0.000} C_DIS
LIN {X 285.996,Y -48.024,Z 165.983,A 170.468,B 90.000,C 0.000} C_DIS
LIN {X 286.010,Y -47.940,Z 166.085,A 170.485,B 90.000,C 0.000} C_DIS
LIN {X 286.044,Y -47.739,Z 166.127,A 170.525,B 90.000,C 0.000} C_DIS
LIN {X 286.051,Y -47.697,Z 166.178,A 170.533,B 90.000,C 0.000} C_DIS
LIN {X 286.061,Y -47.634,Z 166.229,A 170.546,B 90.000,C 0.000} C_DIS
LIN {X 286.111,Y -47.332,Z 166.272,A 170.606,B 90.000,C 0.000} C_DIS
LIN {X 286.122,Y -47.269,Z 166.323,A 170.619,B 90.000,C 0.000} C_DIS
LIN {X 286.129,Y -47.228,Z 166.374,A 170.627,B 90.000,C 0.000} C_DIS
LIN {X 286.162,Y -47.026,Z 166.416,A 170.668,B 90.000,C 0.000} C_DIS
LIN {X 286.175,Y -46.942,Z 166.518,A 170.685,B 90.000,C 0.000} C_DIS
LIN {X 286.208,Y -46.741,Z 166.561,A 170.725,B 90.000,C 0.000} C_DIS
LIN {X 286.215,Y -46.699,Z 166.612,A 170.733,B 90.000,C 0.000} C_DIS
LIN {X 286.226,Y -46.636,Z 166.663,A 170.746,B 90.000,C 0.000} C_DIS
LIN {X 286.275,Y -46.334,Z 166.705,A 170.806,B 90.000,C 0.000} C_DIS
LIN {X 286.285,Y -46.271,Z 166.756,A 170.819,B 90.000,C 0.000} C_DIS
LIN {X 286.292,Y -46.229,Z 166.807,A 170.827,B 90.000,C 0.000} C_DIS
LIN {X 286.324,Y -46.028,Z 166.850,A 170.868,B 90.000,C 0.000} C_DIS
LIN {X 286.338,Y -45.944,Z 166.952,A 170.884,B 90.000,C 0.000} C_DIS
LIN {X 286.370,Y -45.742,Z 166.994,A 170.925,B 90.000,C 0.000} C_DIS
LIN {X 286.376,Y -45.700,Z 167.045,A 170.933,B 90.000,C 0.000} C_DIS
LIN {X 286.387,Y -45.637,Z 167.096,A 170.946,B 90.000,C 0.000} C_DIS
LIN {X 286.435,Y -45.335,Z 167.139,A 171.006,B 90.000,C 0.000} C_DIS
LIN {X 286.444,Y -45.272,Z 167.190,A 171.019,B 90.000,C 0.000} C_DIS
LIN {X 286.451,Y -45.230,Z 167.241,A 171.027,B 90.000,C 0.000} C_DIS
LIN {X 286.483,Y -45.028,Z 167.283,A 171.068,B 90.000,C 0.000} C_DIS
LIN {X 286.496,Y -44.945,Z 167.385,A 171.084,B 90.000,C 0.000} C_DIS
LIN {X 286.528,Y -44.743,Z 167.428,A 171.125,B 90.000,C 0.000} C_DIS
LIN {X 286.534,Y -44.701,Z 167.479,A 171.133,B 90.000,C 0.000} C_DIS
LIN {X 286.544,Y -44.638,Z 167.530,A 171.146,B 90.000,C 0.000} C_DIS
LIN {X 286.591,Y -44.335,Z 167.572,A 171.206,B 90.000,C 0.000} C_DIS
LIN {X 286.601,Y -44.272,Z 167.623,A 171.219,B 90.000,C 0.000} C_DIS
LIN {X 286.607,Y -44.230,Z 167.675,A 171.227,B 90.000,C 0.000} C_DIS
LIN {X 286.638,Y -44.029,Z 167.717,A 171.267,B 90.000,C 0.000} C_DIS
LIN {X 286.651,Y -43.945,Z 167.819,A 171.284,B 90.000,C 0.000} C_DIS
LIN {X 286.682,Y -43.743,Z 167.861,A 171.325,B 90.000,C 0.000} C_DIS
LIN {X 286.688,Y -43.701,Z 167.913,A 171.333,B 90.000,C 0.000} C_DIS
LIN {X 286.698,Y -43.638,Z 167.964,A 171.345,B 90.000,C 0.000} C_DIS
LIN {X 286.744,Y -43.335,Z 168.006,A 171.406,B 90.000,C 0.000} C_DIS
LIN {X 286.753,Y -43.272,Z 168.057,A 171.419,B 90.000,C 0.000} C_DIS
LIN {X 286.760,Y -43.230,Z 168.108,A 171.427,B 90.000,C 0.000} C_DIS
LIN {X 286.790,Y -43.028,Z 168.151,A 171.467,B 90.000,C 0.000} C_DIS
LIN {X 286.803,Y -42.945,Z 168.253,A 171.484,B 90.000,C 0.000} C_DIS
LIN {X 286.833,Y -42.743,Z 168.295,A 171.524,B 90.000,C 0.000} C_DIS
LIN {X 286.839,Y -42.701,Z 168.346,A 171.533,B 90.000,C 0.000} C_DIS
LIN {X 286.848,Y -42.638,Z 168.397,A 171.545,B 90.000,C 0.000} C_DIS
LIN {X 286.893,Y -42.335,Z 168.440,A 171.606,B 90.000,C 0.000} C_DIS
LIN {X 286.903,Y -42.272,Z 168.491,A 171.618,B 90.000,C 0.000} C_DIS
LIN {X 286.909,Y -42.230,Z 168.542,A 171.627,B 90.000,C 0.000} C_DIS
LIN {X 286.938,Y -42.028,Z 168.584,A 171.667,B 90.000,C 0.000} C_DIS
LIN {X 286.951,Y -41.944,Z 168.686,A 171.684,B 90.000,C 0.000} C_DIS
LIN {X 286.980,Y -41.742,Z 168.729,A 171.724,B 90.000,C 0.000} C_DIS
LIN {X 286.986,Y -41.700,Z 168.780,A 171.733,B 90.000,C 0.000} C_DIS
LIN {X 286.995,Y -41.637,Z 168.831,A 171.745,B 90.000,C 0.000} C_DIS
LIN {X 287.039,Y -41.334,Z 168.873,A 171.806,B 90.000,C 0.000} C_DIS
LIN {X 287.048,Y -41.271,Z 168.924,A 171.818,B 90.000,C 0.000} C_DIS
LIN {X 287.054,Y -41.229,Z 168.975,A 171.827,B 90.000,C 0.000} C_DIS
LIN {X 287.083,Y -41.026,Z 169.018,A 171.867,B 90.000,C 0.000} C_DIS
LIN {X 287.095,Y -40.942,Z 169.120,A 171.884,B 90.000,C 0.000} C_DIS
LIN {X 287.124,Y -40.740,Z 169.162,A 171.924,B 90.000,C 0.000} C_DIS
LIN {X 287.130,Y -40.698,Z 169.213,A 171.933,B 90.000,C 0.000} C_DIS
LIN {X 287.139,Y -40.635,Z 169.264,A 171.945,B 90.000,C 0.000} C_DIS
LIN {X 287.182,Y -40.332,Z 169.307,A 172.006,B 90.000,C 0.000} C_DIS
LIN {X 287.191,Y -40.269,Z 169.358,A 172.018,B 90.000,C 0.000} C_DIS
LIN {X 287.196,Y -40.227,Z 169.409,A 172.027,B 90.000,C 0.000} C_DIS
LIN {X 287.225,Y -40.025,Z 169.451,A 172.067,B 90.000,C 0.000} C_DIS
LIN {X 287.236,Y -39.941,Z 169.553,A 172.084,B 90.000,C 0.000} C_DIS
LIN {X 287.264,Y -39.738,Z 169.596,A 172.124,B 90.000,C 0.000} C_DIS
LIN {X 287.270,Y -39.696,Z 169.647,A 172.132,B 90.000,C 0.000} C_DIS
LIN {X 287.279,Y -39.633,Z 169.698,A 172.145,B 90.000,C 0.000} C_DIS
LIN {X 287.321,Y -39.330,Z 169.740,A 172.206,B 90.000,C 0.000} C_DIS
LIN {X 287.329,Y -39.267,Z 169.791,A 172.218,B 90.000,C 0.000} C_DIS
LIN {X 287.335,Y -39.225,Z 169.842,A 172.226,B 90.000,C 0.000} C_DIS
LIN {X 287.363,Y -39.022,Z 169.885,A 172.267,B 90.000,C 0.000} C_DIS
LIN {X 287.374,Y -38.938,Z 169.987,A 172.284,B 90.000,C 0.000} C_DIS
LIN {X 287.401,Y -38.736,Z 170.029,A 172.324,B 90.000,C 0.000} C_DIS
LIN {X 287.407,Y -38.694,Z 170.080,A 172.332,B 90.000,C 0.000} C_DIS
LIN {X 287.415,Y -38.631,Z 170.131,A 172.345,B 90.000,C 0.000} C_DIS
LIN {X 287.456,Y -38.327,Z 170.174,A 172.405,B 90.000,C 0.000} C_DIS
LIN {X 287.465,Y -38.264,Z 170.225,A 172.418,B 90.000,C 0.000} C_DIS
LIN {X 287.470,Y -38.222,Z 170.276,A 172.426,B 90.000,C 0.000} C_DIS
LIN {X 287.497,Y -38.020,Z 170.318,A 172.467,B 90.000,C 0.000} C_DIS
LIN {X 287.508,Y -37.936,Z 170.421,A 172.483,B 90.000,C 0.000} C_DIS
LIN {X 287.535,Y -37.733,Z 170.463,A 172.524,B 90.000,C 0.000} C_DIS
LIN {X 287.540,Y -37.691,Z 170.514,A 172.532,B 90.000,C 0.000} C_DIS
LIN {X 287.549,Y -37.628,Z 170.565,A 172.545,B 90.000,C 0.000} C_DIS
LIN {X 287.588,Y -37.324,Z 170.608,A 172.605,B 90.000,C 0.000} C_DIS
LIN {X 287.596,Y -37.261,Z 170.659,A 172.618,B 90.000,C 0.000} C_DIS
LIN {X 287.602,Y -37.219,Z 170.710,A 172.626,B 90.000,C 0.000} C_DIS
LIN {X 287.628,Y -37.016,Z 170.752,A 172.667,B 90.000,C 0.000} C_DIS
LIN {X 287.639,Y -36.932,Z 170.854,A 172.683,B 90.000,C 0.000} C_DIS
LIN {X 287.665,Y -36.730,Z 170.897,A 172.724,B 90.000,C 0.000} C_DIS
LIN {X 287.670,Y -36.688,Z 170.948,A 172.732,B 90.000,C 0.000} C_DIS
LIN {X 287.678,Y -36.625,Z 170.999,A 172.745,B 90.000,C 0.000} C_DIS
LIN {X 287.717,Y -36.321,Z 171.041,A 172.805,B 90.000,C 0.000} C_DIS
LIN {X 287.725,Y -36.258,Z 171.092,A 172.818,B 90.000,C 0.000} C_DIS
LIN {X 287.730,Y -36.215,Z 171.143,A 172.826,B 90.000,C 0.000} C_DIS
LIN {X 287.755,Y -36.013,Z 171.186,A 172.866,B 90.000,C 0.000} C_DIS
LIN {X 287.766,Y -35.929,Z 171.288,A 172.883,B 90.000,C 0.000} C_DIS
LIN {X 287.791,Y -35.726,Z 171.330,A 172.924,B 90.000,C 0.000} C_DIS
LIN {X 287.796,Y -35.684,Z 171.381,A 172.932,B 90.000,C 0.000} C_DIS
LIN {X 287.804,Y -35.621,Z 171.432,A 172.945,B 90.000,C 0.000} C_DIS
LIN {X 287.841,Y -35.317,Z 171.475,A 173.005,B 90.000,C 0.000} C_DIS
LIN {X 287.849,Y -35.254,Z 171.526,A 173.018,B 90.000,C 0.000} C_DIS
LIN {X 287.854,Y -35.211,Z 171.577,A 173.026,B 90.000,C 0.000} C_DIS
LIN {X 287.879,Y -35.009,Z 171.619,A 173.066,B 90.000,C 0.000} C_DIS
LIN {X 287.889,Y -34.924,Z 171.721,A 173.083,B 90.000,C 0.000} C_DIS
LIN {X 287.914,Y -34.722,Z 171.764,A 173.123,B 90.000,C 0.000} C_DIS
LIN {X 287.919,Y -34.680,Z 171.815,A 173.132,B 90.000,C 0.000} C_DIS
LIN {X 287.927,Y -34.616,Z 171.866,A 173.144,B 90.000,C 0.000} C_DIS
LIN {X 287.963,Y -34.312,Z 171.908,A 173.205,B 90.000,C 0.000} C_DIS
LIN {X 287.970,Y -34.249,Z 171.959,A 173.218,B 90.000,C 0.000} C_DIS
LIN {X 287.975,Y -34.207,Z 172.010,A 173.226,B 90.000,C 0.000} C_DIS
LIN {X 287.999,Y -34.004,Z 172.053,A 173.266,B 90.000,C 0.000} C_DIS
LIN {X 288.009,Y -33.920,Z 172.155,A 173.283,B 90.000,C 0.000} C_DIS
LIN {X 288.033,Y -33.717,Z 172.197,A 173.323,B 90.000,C 0.000} C_DIS
LIN {X 288.038,Y -33.675,Z 172.248,A 173.332,B 90.000,C 0.000} C_DIS
LIN {X 288.046,Y -33.612,Z 172.299,A 173.344,B 90.000,C 0.000} C_DIS
LIN {X 288.081,Y -33.308,Z 172.342,A 173.405,B 90.000,C 0.000} C_DIS
LIN {X 288.088,Y -33.244,Z 172.393,A 173.417,B 90.000,C 0.000} C_DIS
LIN {X 288.093,Y -33.202,Z 172.444,A 173.426,B 90.000,C 0.000} C_DIS
LIN {X 288.116,Y -32.999,Z 172.486,A 173.466,B 90.000,C 0.000} C_DIS
LIN {X 288.126,Y -32.915,Z 172.588,A 173.483,B 90.000,C 0.000} C_DIS
LIN {X 288.149,Y -32.712,Z 172.631,A 173.523,B 90.000,C 0.000} C_DIS
LIN {X 288.159,Y -32.628,Z 172.733,A 173.540,B 90.000,C 0.000} C_DIS
LIN {X 288.182,Y -32.425,Z 172.775,A 173.580,B 90.000,C 0.000} C_DIS
LIN {X 288.186,Y -32.383,Z 172.826,A 173.589,B 90.000,C 0.000} C_DIS
LIN {X 288.193,Y -32.319,Z 172.878,A 173.601,B 90.000,C 0.000} C_DIS
LIN {X 288.227,Y -32.015,Z 172.920,A 173.662,B 90.000,C 0.000} C_DIS
LIN {X 288.234,Y -31.952,Z 172.971,A 173.674,B 90.000,C 0.000} C_DIS
LIN {X 288.239,Y -31.910,Z 173.022,A 173.683,B 90.000,C 0.000} C_DIS
LIN {X 288.261,Y -31.707,Z 173.064,A 173.723,B 90.000,C 0.000} C_DIS
LIN {X 288.266,Y -31.665,Z 173.116,A 173.731,B 90.000,C 0.000} C_DIS
LIN {X 288.273,Y -31.601,Z 173.167,A 173.744,B 90.000,C 0.000} C_DIS
LIN {X 288.306,Y -31.297,Z 173.209,A 173.805,B 90.000,C 0.000} C_DIS
LIN {X 288.313,Y -31.233,Z 173.260,A 173.817,B 90.000,C 0.000} C_DIS
LIN {X 288.318,Y -31.191,Z 173.311,A 173.826,B 90.000,C 0.000} C_DIS
LIN {X 288.340,Y -30.988,Z 173.354,A 173.866,B 90.000,C 0.000} C_DIS
LIN {X 288.349,Y -30.904,Z 173.456,A 173.883,B 90.000,C 0.000} C_DIS
LIN {X 288.370,Y -30.701,Z 173.498,A 173.923,B 90.000,C 0.000} C_DIS
LIN {X 288.375,Y -30.659,Z 173.549,A 173.931,B 90.000,C 0.000} C_DIS
LIN {X 288.382,Y -30.595,Z 173.600,A 173.944,B 90.000,C 0.000} C_DIS
LIN {X 288.414,Y -30.291,Z 173.643,A 174.004,B 90.000,C 0.000} C_DIS
LIN {X 288.420,Y -30.227,Z 173.694,A 174.017,B 90.000,C 0.000} C_DIS
LIN {X 288.425,Y -30.185,Z 173.745,A 174.025,B 90.000,C 0.000} C_DIS
LIN {X 288.446,Y -29.982,Z 173.787,A 174.066,B 90.000,C 0.000} C_DIS
LIN {X 288.455,Y -29.898,Z 173.889,A 174.083,B 90.000,C 0.000} C_DIS
LIN {X 288.476,Y -29.695,Z 173.932,A 174.123,B 90.000,C 0.000} C_DIS
LIN {X 288.484,Y -29.610,Z 174.034,A 174.140,B 90.000,C 0.000} C_DIS
LIN {X 288.505,Y -29.407,Z 174.076,A 174.180,B 90.000,C 0.000} C_DIS
LIN {X 288.509,Y -29.365,Z 174.127,A 174.188,B 90.000,C 0.000} C_DIS
LIN {X 288.516,Y -29.302,Z 174.178,A 174.201,B 90.000,C 0.000} C_DIS
LIN {X 288.547,Y -28.997,Z 174.221,A 174.261,B 90.000,C 0.000} C_DIS
LIN {X 288.553,Y -28.934,Z 174.272,A 174.274,B 90.000,C 0.000} C_DIS
LIN {X 288.557,Y -28.891,Z 174.323,A 174.282,B 90.000,C 0.000} C_DIS
LIN {X 288.578,Y -28.688,Z 174.365,A 174.323,B 90.000,C 0.000} C_DIS
LIN {X 288.582,Y -28.646,Z 174.416,A 174.331,B 90.000,C 0.000} C_DIS
LIN {X 288.588,Y -28.582,Z 174.467,A 174.344,B 90.000,C 0.000} C_DIS
LIN {X 288.618,Y -28.278,Z 174.510,A 174.404,B 90.000,C 0.000} C_DIS
LIN {X 288.624,Y -28.214,Z 174.561,A 174.417,B 90.000,C 0.000} C_DIS
LIN {X 288.628,Y -28.172,Z 174.612,A 174.425,B 90.000,C 0.000} C_DIS
LIN {X 288.648,Y -27.969,Z 174.654,A 174.466,B 90.000,C 0.000} C_DIS
LIN {X 288.656,Y -27.884,Z 174.756,A 174.482,B 90.000,C 0.000} C_DIS
LIN {X 288.676,Y -27.681,Z 174.799,A 174.523,B 90.000,C 0.000} C_DIS
LIN {X 288.684,Y -27.597,Z 174.901,A 174.539,B 90.000,C 0.000} C_DIS
LIN {X 288.703,Y -27.393,Z 174.943,A 174.580,B 90.000,C 0.000} C_DIS
LIN {X 288.707,Y -27.351,Z 174.994,A 174.588,B 90.000,C 0.000} C_DIS
LIN {X 288.713,Y -27.288,Z 175.045,A 174.601,B 90.000,C 0.000} C_DIS
LIN {X 288.742,Y -26.983,Z 175.088,A 174.661,B 90.000,C 0.000} C_DIS
LIN {X 288.748,Y -26.920,Z 175.139,A 174.674,B 90.000,C 0.000} C_DIS
LIN {X 288.752,Y -26.877,Z 175.190,A 174.682,B 90.000,C 0.000} C_DIS
LIN {X 288.771,Y -26.674,Z 175.232,A 174.723,B 90.000,C 0.000} C_DIS
LIN {X 288.778,Y -26.589,Z 175.334,A 174.739,B 90.000,C 0.000} C_DIS
LIN {X 288.797,Y -26.386,Z 175.377,A 174.780,B 90.000,C 0.000} C_DIS
LIN {X 288.801,Y -26.344,Z 175.428,A 174.788,B 90.000,C 0.000} C_DIS
LIN {X 288.807,Y -26.280,Z 175.479,A 174.801,B 90.000,C 0.000} C_DIS
LIN {X 288.834,Y -25.975,Z 175.521,A 174.861,B 90.000,C 0.000} C_DIS
LIN {X 288.840,Y -25.912,Z 175.573,A 174.874,B 90.000,C 0.000} C_DIS
LIN {X 288.844,Y -25.870,Z 175.624,A 174.882,B 90.000,C 0.000} C_DIS
LIN {X 288.862,Y -25.666,Z 175.666,A 174.922,B 90.000,C 0.000} C_DIS
LIN {X 288.869,Y -25.582,Z 175.768,A 174.939,B 90.000,C 0.000} C_DIS
LIN {X 288.887,Y -25.378,Z 175.811,A 174.980,B 90.000,C 0.000} C_DIS
LIN {X 288.891,Y -25.336,Z 175.862,A 174.988,B 90.000,C 0.000} C_DIS
LIN {X 288.897,Y -25.273,Z 175.913,A 175.000,B 90.000,C 0.000} C_DIS
LIN {X 288.923,Y -24.968,Z 175.955,A 175.061,B 90.000,C 0.000} C_DIS
LIN {X 288.929,Y -24.904,Z 176.006,A 175.074,B 90.000,C 0.000} C_DIS
LIN {X 288.932,Y -24.862,Z 176.057,A 175.082,B 90.000,C 0.000} C_DIS
LIN {X 288.950,Y -24.659,Z 176.100,A 175.122,B 90.000,C 0.000} C_DIS
LIN {X 288.957,Y -24.574,Z 176.202,A 175.139,B 90.000,C 0.000} C_DIS
LIN {X 288.974,Y -24.370,Z 176.244,A 175.179,B 90.000,C 0.000} C_DIS
LIN {X 288.978,Y -24.328,Z 176.295,A 175.188,B 90.000,C 0.000} C_DIS
LIN {X 288.983,Y -24.265,Z 176.346,A 175.200,B 90.000,C 0.000} C_DIS
LIN {X 289.009,Y -23.960,Z 176.389,A 175.261,B 90.000,C 0.000} C_DIS
LIN {X 289.014,Y -23.896,Z 176.440,A 175.273,B 90.000,C 0.000} C_DIS
LIN {X 289.017,Y -23.854,Z 176.491,A 175.282,B 90.000,C 0.000} C_DIS
LIN {X 289.034,Y -23.650,Z 176.533,A 175.322,B 90.000,C 0.000} C_DIS
LIN {X 289.041,Y -23.566,Z 176.635,A 175.339,B 90.000,C 0.000} C_DIS
LIN {X 289.057,Y -23.362,Z 176.678,A 175.379,B 90.000,C 0.000} C_DIS
LIN {X 289.061,Y -23.320,Z 176.729,A 175.388,B 90.000,C 0.000} C_DIS
LIN {X 289.063,Y -23.287,Z 176.780,A 175.394,B 90.000,C 0.000} C_DIS
LIN {X 289.070,Y -23.209,Z 176.801,A 175.410,B 90.000,C 0.000} C_DIS
LIN {X 289.080,Y -23.078,Z 176.853,A 175.436,B 90.000,C 0.000} C_DIS
LIN {X 289.093,Y -22.920,Z 176.978,A 175.467,B 90.000,C 0.000} C_DIS
LIN {X 289.107,Y -22.744,Z 177.156,A 175.502,B 90.000,C 0.000} C_DIS
LIN {X 289.107,Y -22.746,Z 179.656,A 175.501,B 90.000,C 0.000} C_DIS
LIN {X 289.101,Y -22.816,Z 181.715,A 175.488,B 90.000,C 0.000} C_DIS
LIN {X 289.097,Y -22.868,Z 181.923,A 175.477,B 90.000,C 0.000} C_DIS
LIN {X 289.095,Y -22.888,Z 183.237,A 175.473,B 90.000,C 0.000} C_DIS
LIN {X 289.076,Y -23.137,Z 183.488,A 175.424,B 90.000,C 0.000} C_DIS
LIN {X 289.054,Y -23.401,Z 183.693,A 175.372,B 90.000,C 0.000} C_DIS
LIN {X 289.029,Y -23.714,Z 183.738,A 175.310,B 90.000,C 0.000} C_DIS
LIN {X 289.010,Y -23.944,Z 183.717,A 175.264,B 90.000,C 0.000} C_DIS
LIN {X 289.002,Y -24.040,Z 183.666,A 175.245,B 90.000,C 0.000} C_DIS
LIN {X 288.997,Y -24.104,Z 183.615,A 175.232,B 90.000,C 0.000} C_DIS
LIN {X 288.971,Y -24.409,Z 183.573,A 175.172,B 90.000,C 0.000} C_DIS
LIN {X 288.960,Y -24.536,Z 183.471,A 175.147,B 90.000,C 0.000} C_DIS
LIN {X 288.934,Y -24.841,Z 183.428,A 175.086,B 90.000,C 0.000} C_DIS
LIN {X 288.929,Y -24.904,Z 183.377,A 175.074,B 90.000,C 0.000} C_DIS
LIN {X 288.925,Y -24.946,Z 183.326,A 175.065,B 90.000,C 0.000} C_DIS
LIN {X 288.907,Y -25.150,Z 183.284,A 175.025,B 90.000,C 0.000} C_DIS
LIN {X 288.900,Y -25.234,Z 183.182,A 175.008,B 90.000,C 0.000} C_DIS
LIN {X 288.891,Y -25.336,Z 183.160,A 174.988,B 90.000,C 0.000} C_DIS
LIN {X 288.882,Y -25.438,Z 183.182,A 174.968,B 90.000,C 0.000} C_DIS
LIN {X 288.878,Y -25.480,Z 183.233,A 174.959,B 90.000,C 0.000} C_DIS
LIN {X 288.882,Y -25.438,Z 183.284,A 174.968,B 90.000,C 0.000} C_DIS
LIN {X 288.900,Y -25.234,Z 183.326,A 175.008,B 90.000,C 0.000} C_DIS
LIN {X 288.907,Y -25.150,Z 183.428,A 175.025,B 90.000,C 0.000} C_DIS
LIN {X 288.925,Y -24.946,Z 183.471,A 175.065,B 90.000,C 0.000} C_DIS
LIN {X 288.932,Y -24.862,Z 183.573,A 175.082,B 90.000,C 0.000} C_DIS
LIN {X 288.950,Y -24.658,Z 183.615,A 175.122,B 90.000,C 0.000} C_DIS
LIN {X 288.957,Y -24.574,Z 183.717,A 175.139,B 90.000,C 0.000} C_DIS
LIN {X 288.974,Y -24.370,Z 183.760,A 175.179,B 90.000,C 0.000} C_DIS
LIN {X 288.981,Y -24.286,Z 183.862,A 175.196,B 90.000,C 0.000} C_DIS
LIN {X 288.998,Y -24.082,Z 183.904,A 175.237,B 90.000,C 0.000} C_DIS
LIN {X 289.005,Y -23.998,Z 184.006,A 175.253,B 90.000,C 0.000} C_DIS
LIN {X 289.022,Y -23.794,Z 184.049,A 175.294,B 90.000,C 0.000} C_DIS
LIN {X 289.026,Y -23.752,Z 184.100,A 175.302,B 90.000,C 0.000} C_DIS
LIN {X 289.031,Y -23.689,Z 184.151,A 175.315,B 90.000,C 0.000} C_DIS
LIN {X 289.056,Y -23.383,Z 184.193,A 175.375,B 90.000,C 0.000} C_DIS
LIN {X 289.061,Y -23.320,Z 184.244,A 175.388,B 90.000,C 0.000} C_DIS
LIN {X 289.064,Y -23.277,Z 184.295,A 175.396,B 90.000,C 0.000} C_DIS
LIN {X 289.081,Y -23.074,Z 184.338,A 175.436,B 90.000,C 0.000} C_DIS
LIN {X 289.087,Y -22.989,Z 184.440,A 175.453,B 90.000,C 0.000} C_DIS
LIN {X 289.103,Y -22.786,Z 184.482,A 175.494,B 90.000,C 0.000} C_DIS
LIN {X 289.110,Y -22.701,Z 184.584,A 175.510,B 90.000,C 0.000} C_DIS
LIN {X 289.126,Y -22.498,Z 184.627,A 175.551,B 90.000,C 0.000} C_DIS
LIN {X 289.133,Y -22.413,Z 184.729,A 175.567,B 90.000,C 0.000} C_DIS
LIN {X 289.148,Y -22.209,Z 184.771,A 175.608,B 90.000,C 0.000} C_DIS
LIN {X 289.154,Y -22.129,Z 184.873,A 175.624,B 90.000,C 0.000} C_DIS
LIN {X 289.161,Y -22.039,Z 184.895,A 175.642,B 90.000,C 0.000} C_DIS
LIN {X 289.171,Y -21.918,Z 184.937,A 175.666,B 90.000,C 0.000} C_DIS
LIN {X 289.179,Y -21.807,Z 185.039,A 175.688,B 90.000,C 0.000} C_DIS
LIN {X 289.207,Y -21.438,Z 185.283,A 175.761,B 90.000,C 0.000} C_DIS
LIN {X 289.241,Y -20.967,Z 185.766,A 175.854,B 90.000,C 0.000} C_DIS
LIN {X 289.248,Y -20.870,Z 185.941,A 175.873,B 90.000,C 0.000} C_DIS
LIN {X 289.250,Y -20.849,Z 186.018,A 175.877,B 90.000,C 0.000} C_DIS
LIN {X 289.253,Y -20.798,Z 186.051,A 175.887,B 90.000,C 0.000} C_DIS
LIN {X 289.257,Y -20.747,Z 186.093,A 175.897,B 90.000,C 0.000} C_DIS
LIN {X 289.260,Y -20.705,Z 186.297,A 175.906,B 90.000,C 0.000} C_DIS
LIN {X 289.264,Y -20.654,Z 186.340,A 175.916,B 90.000,C 0.000} C_DIS
LIN {X 289.267,Y -20.602,Z 186.521,A 175.926,B 90.000,C 0.000} C_DIS
LIN {X 289.267,Y -20.602,Z 187.460,A 175.926,B 90.000,C 0.000} C_DIS
LIN {X 289.264,Y -20.654,Z 187.641,A 175.916,B 90.000,C 0.000} C_DIS
LIN {X 289.260,Y -20.705,Z 187.673,A 175.906,B 90.000,C 0.000} C_DIS
LIN {X 289.258,Y -20.726,Z 187.751,A 175.902,B 90.000,C 0.000} C_DIS
LIN {X 289.251,Y -20.824,Z 187.930,A 175.882,B 90.000,C 0.000} C_DIS
LIN {X 289.235,Y -21.050,Z 188.183,A 175.838,B 90.000,C 0.000} C_DIS
LIN {X 289.217,Y -21.302,Z 188.410,A 175.787,B 90.000,C 0.000} C_DIS
LIN {X 289.203,Y -21.481,Z 188.508,A 175.752,B 90.000,C 0.000} C_DIS
LIN {X 289.198,Y -21.558,Z 188.529,A 175.737,B 90.000,C 0.000} C_DIS
LIN {X 289.195,Y -21.591,Z 188.580,A 175.730,B 90.000,C 0.000} C_DIS
LIN {X 289.186,Y -21.715,Z 188.631,A 175.706,B 90.000,C 0.000} C_DIS
LIN {X 289.138,Y -22.343,Z 188.676,A 175.581,B 90.000,C 0.000} C_DIS
LIN {X 289.127,Y -22.485,Z 188.743,A 175.553,B 90.000,C 0.000} C_DIS
LIN {X 289.124,Y -22.527,Z 188.797,A 175.545,B 90.000,C 0.000} C_DIS
LIN {X 289.120,Y -22.569,Z 188.743,A 175.536,B 90.000,C 0.000} C_DIS
LIN {X 289.109,Y -22.712,Z 188.676,A 175.508,B 90.000,C 0.000} C_DIS
LIN {X 289.059,Y -23.339,Z 188.631,A 175.384,B 90.000,C 0.000} C_DIS
LIN {X 289.049,Y -23.464,Z 188.580,A 175.359,B 90.000,C 0.000} C_DIS
LIN {X 289.044,Y -23.527,Z 188.529,A 175.347,B 90.000,C 0.000} C_DIS
LIN {X 289.019,Y -23.833,Z 188.487,A 175.286,B 90.000,C 0.000} C_DIS
LIN {X 289.009,Y -23.959,Z 188.385,A 175.261,B 90.000,C 0.000} C_DIS
LIN {X 288.983,Y -24.265,Z 188.342,A 175.200,B 90.000,C 0.000} C_DIS
LIN {X 288.978,Y -24.328,Z 188.291,A 175.188,B 90.000,C 0.000} C_DIS
LIN {X 288.971,Y -24.413,Z 188.240,A 175.171,B 90.000,C 0.000} C_DIS
LIN {X 288.936,Y -24.820,Z 188.198,A 175.090,B 90.000,C 0.000} C_DIS
LIN {X 288.929,Y -24.904,Z 188.147,A 175.074,B 90.000,C 0.000} C_DIS
LIN {X 288.923,Y -24.968,Z 188.095,A 175.061,B 90.000,C 0.000} C_DIS
LIN {X 288.897,Y -25.273,Z 188.053,A 175.000,B 90.000,C 0.000} C_DIS
LIN {X 288.891,Y -25.336,Z 188.002,A 174.988,B 90.000,C 0.000} C_DIS
LIN {X 288.884,Y -25.421,Z 187.951,A 174.971,B 90.000,C 0.000} C_DIS
LIN {X 288.848,Y -25.827,Z 187.908,A 174.890,B 90.000,C 0.000} C_DIS
LIN {X 288.840,Y -25.912,Z 187.857,A 174.874,B 90.000,C 0.000} C_DIS
LIN {X 288.834,Y -25.975,Z 187.806,A 174.861,B 90.000,C 0.000} C_DIS
LIN {X 288.807,Y -26.280,Z 187.764,A 174.801,B 90.000,C 0.000} C_DIS
LIN {X 288.801,Y -26.344,Z 187.713,A 174.788,B 90.000,C 0.000} C_DIS
LIN {X 288.793,Y -26.428,Z 187.662,A 174.771,B 90.000,C 0.000} C_DIS
LIN {X 288.756,Y -26.835,Z 187.619,A 174.691,B 90.000,C 0.000} C_DIS
LIN {X 288.748,Y -26.919,Z 187.568,A 174.674,B 90.000,C 0.000} C_DIS
LIN {X 288.743,Y -26.974,Z 187.517,A 174.663,B 90.000,C 0.000} C_DIS
LIN {X 288.731,Y -27.105,Z 187.496,A 174.637,B 90.000,C 0.000} C_DIS
LIN {X 288.711,Y -27.313,Z 187.569,A 174.596,B 90.000,C 0.000} C_DIS
LIN {X 288.607,Y -28.390,Z 188.444,A 174.382,B 90.000,C 0.000} C_DIS
LIN {X 288.593,Y -28.531,Z 188.508,A 174.354,B 90.000,C 0.000} C_DIS
LIN {X 288.585,Y -28.612,Z 188.529,A 174.338,B 90.000,C 0.000} C_DIS
LIN {X 288.582,Y -28.646,Z 188.580,A 174.331,B 90.000,C 0.000} C_DIS
LIN {X 288.578,Y -28.688,Z 188.631,A 174.323,B 90.000,C 0.000} C_DIS
LIN {X 288.557,Y -28.891,Z 188.674,A 174.282,B 90.000,C 0.000} C_DIS
LIN {X 288.549,Y -28.976,Z 188.776,A 174.266,B 90.000,C 0.000} C_DIS
LIN {X 288.528,Y -29.179,Z 188.818,A 174.225,B 90.000,C 0.000} C_DIS
LIN {X 288.520,Y -29.263,Z 188.920,A 174.209,B 90.000,C 0.000} C_DIS
LIN {X 288.499,Y -29.466,Z 188.963,A 174.168,B 90.000,C 0.000} C_DIS
LIN {X 288.495,Y -29.509,Z 189.014,A 174.160,B 90.000,C 0.000} C_DIS
LIN {X 288.486,Y -29.593,Z 189.065,A 174.143,B 90.000,C 0.000} C_DIS
LIN {X 288.444,Y -29.999,Z 189.107,A 174.062,B 90.000,C 0.000} C_DIS
LIN {X 288.427,Y -30.168,Z 189.209,A 174.029,B 90.000,C 0.000} C_DIS
LIN {X 288.384,Y -30.574,Z 189.252,A 173.948,B 90.000,C 0.000} C_DIS
LIN {X 288.375,Y -30.659,Z 189.303,A 173.931,B 90.000,C 0.000} C_DIS
LIN {X 288.344,Y -30.946,Z 189.356,A 173.874,B 90.000,C 0.000} C_DIS
LIN {X 288.170,Y -32.526,Z 189.356,A 173.560,B 90.000,C 0.000} C_DIS
LIN {X 288.138,Y -32.813,Z 189.303,A 173.503,B 90.000,C 0.000} C_DIS
LIN {X 288.128,Y -32.898,Z 189.252,A 173.486,B 90.000,C 0.000} C_DIS
LIN {X 288.081,Y -33.303,Z 189.209,A 173.406,B 90.000,C 0.000} C_DIS
LIN {X 288.072,Y -33.388,Z 189.158,A 173.389,B 90.000,C 0.000} C_DIS
LIN {X 288.064,Y -33.451,Z 189.107,A 173.376,B 90.000,C 0.000} C_DIS
LIN {X 288.029,Y -33.755,Z 189.065,A 173.316,B 90.000,C 0.000} C_DIS
LIN {X 288.014,Y -33.882,Z 188.963,A 173.291,B 90.000,C 0.000} C_DIS
LIN {X 287.978,Y -34.186,Z 188.920,A 173.230,B 90.000,C 0.000} C_DIS
LIN {X 287.970,Y -34.249,Z 188.869,A 173.218,B 90.000,C 0.000} C_DIS
LIN {X 287.965,Y -34.291,Z 188.818,A 173.209,B 90.000,C 0.000} C_DIS
LIN {X 287.941,Y -34.494,Z 188.776,A 173.169,B 90.000,C 0.000} C_DIS
LIN {X 287.932,Y -34.574,Z 188.674,A 173.153,B 90.000,C 0.000} C_DIS
LIN {X 287.921,Y -34.664,Z 188.652,A 173.135,B 90.000,C 0.000} C_DIS
LIN {X 287.906,Y -34.784,Z 188.610,A 173.111,B 90.000,C 0.000} C_DIS
LIN {X 287.880,Y -35.001,Z 188.406,A 173.068,B 90.000,C 0.000} C_DIS
LIN {X 287.853,Y -35.219,Z 188.321,A 173.024,B 90.000,C 0.000} C_DIS
LIN {X 287.840,Y -35.325,Z 188.219,A 173.003,B 90.000,C 0.000} C_DIS
LIN {X 287.791,Y -35.729,Z 187.931,A 172.923,B 90.000,C 0.000} C_DIS
LIN {X 287.706,Y -36.400,Z 187.263,A 172.789,B 90.000,C 0.000} C_DIS
LIN {X 287.641,Y -36.911,Z 186.597,A 172.688,B 90.000,C 0.000} C_DIS
LIN {X 287.633,Y -36.974,Z 186.455,A 172.675,B 90.000,C 0.000} C_DIS
LIN {X 287.631,Y -36.995,Z 186.374,A 172.671,B 90.000,C 0.000} C_DIS
LIN {X 287.624,Y -37.046,Z 186.340,A 172.661,B 90.000,C 0.000} C_DIS
LIN {X 287.618,Y -37.097,Z 186.297,A 172.651,B 90.000,C 0.000} C_DIS
LIN {X 287.612,Y -37.139,Z 186.093,A 172.642,B 90.000,C 0.000} C_DIS
LIN {X 287.599,Y -37.240,Z 186.008,A 172.622,B 90.000,C 0.000} C_DIS
LIN {X 287.594,Y -37.282,Z 185.804,A 172.614,B 90.000,C 0.000} C_DIS
LIN {X 287.580,Y -37.383,Z 185.719,A 172.594,B 90.000,C 0.000} C_DIS
LIN {X 287.575,Y -37.425,Z 185.515,A 172.585,B 90.000,C 0.000} C_DIS
LIN {X 287.568,Y -37.476,Z 185.473,A 172.575,B 90.000,C 0.000} C_DIS
LIN {X 287.562,Y -37.527,Z 185.409,A 172.565,B 90.000,C 0.000} C_DIS
LIN {X 287.556,Y -37.569,Z 185.103,A 172.557,B 90.000,C 0.000} C_DIS
LIN {X 287.550,Y -37.619,Z 185.039,A 172.546,B 90.000,C 0.000} C_DIS
LIN {X 287.543,Y -37.670,Z 184.954,A 172.536,B 90.000,C 0.000} C_DIS
LIN {X 287.537,Y -37.712,Z 184.546,A 172.528,B 90.000,C 0.000} C_DIS
LIN {X 287.531,Y -37.763,Z 184.461,A 172.518,B 90.000,C 0.000} C_DIS
LIN {X 287.524,Y -37.815,Z 184.136,A 172.507,B 90.000,C 0.000} C_DIS
LIN {X 287.524,Y -37.815,Z 182.329,A 172.507,B 90.000,C 0.000} C_DIS
LIN {X 287.531,Y -37.763,Z 182.004,A 172.518,B 90.000,C 0.000} C_DIS
LIN {X 287.537,Y -37.712,Z 181.919,A 172.528,B 90.000,C 0.000} C_DIS
LIN {X 287.543,Y -37.670,Z 181.511,A 172.536,B 90.000,C 0.000} C_DIS
LIN {X 287.550,Y -37.619,Z 181.426,A 172.546,B 90.000,C 0.000} C_DIS
LIN {X 287.556,Y -37.569,Z 181.362,A 172.557,B 90.000,C 0.000} C_DIS
LIN {X 287.562,Y -37.527,Z 181.056,A 172.565,B 90.000,C 0.000} C_DIS
LIN {X 287.568,Y -37.476,Z 180.992,A 172.575,B 90.000,C 0.000} C_DIS
LIN {X 287.575,Y -37.425,Z 180.950,A 172.585,B 90.000,C 0.000} C_DIS
LIN {X 287.580,Y -37.383,Z 180.746,A 172.594,B 90.000,C 0.000} C_DIS
LIN {X 287.594,Y -37.282,Z 180.661,A 172.614,B 90.000,C 0.000} C_DIS
LIN {X 287.599,Y -37.240,Z 180.457,A 172.622,B 90.000,C 0.000} C_DIS
LIN {X 287.612,Y -37.139,Z 180.372,A 172.642,B 90.000,C 0.000} C_DIS
LIN {X 287.618,Y -37.097,Z 180.168,A 172.651,B 90.000,C 0.000} C_DIS
LIN {X 287.631,Y -36.995,Z 180.087,A 172.671,B 90.000,C 0.000} C_DIS
LIN {X 287.633,Y -36.974,Z 179.997,A 172.675,B 90.000,C 0.000} C_DIS
LIN {X 287.639,Y -36.932,Z 179.875,A 172.683,B 90.000,C 0.000} C_DIS
LIN {X 287.665,Y -36.730,Z 179.660,A 172.724,B 90.000,C 0.000} C_DIS
LIN {X 287.670,Y -36.688,Z 179.558,A 172.732,B 90.000,C 0.000} C_DIS
LIN {X 287.689,Y -36.536,Z 179.323,A 172.762,B 90.000,C 0.000} C_DIS
LIN {X 287.703,Y -36.428,Z 179.195,A 172.784,B 90.000,C 0.000} C_DIS
LIN {X 287.694,Y -36.495,Z 179.080,A 172.770,B 90.000,C 0.000} C_DIS
LIN {X 287.678,Y -36.627,Z 179.002,A 172.744,B 90.000,C 0.000} C_DIS
LIN {X 287.640,Y -36.920,Z 178.948,A 172.686,B 90.000,C 0.000} C_DIS
LIN {X 287.625,Y -37.037,Z 178.846,A 172.662,B 90.000,C 0.000} C_DIS
LIN {X 287.586,Y -37.341,Z 178.803,A 172.602,B 90.000,C 0.000} C_DIS
LIN {X 287.578,Y -37.404,Z 178.752,A 172.589,B 90.000,C 0.000} C_DIS
LIN {X 287.572,Y -37.446,Z 178.701,A 172.581,B 90.000,C 0.000} C_DIS
LIN {X 287.546,Y -37.649,Z 178.659,A 172.541,B 90.000,C 0.000} C_DIS
LIN {X 287.540,Y -37.691,Z 178.608,A 172.532,B 90.000,C 0.000} C_DIS
LIN {X 287.532,Y -37.754,Z 178.557,A 172.520,B 90.000,C 0.000} C_DIS
LIN {X 287.492,Y -38.058,Z 178.514,A 172.459,B 90.000,C 0.000} C_DIS
LIN {X 287.475,Y -38.184,Z 178.412,A 172.434,B 90.000,C 0.000} C_DIS
LIN {X 287.435,Y -38.487,Z 178.370,A 172.373,B 90.000,C 0.000} C_DIS
LIN {X 287.418,Y -38.614,Z 178.268,A 172.348,B 90.000,C 0.000} C_DIS
LIN {X 287.377,Y -38.917,Z 178.225,A 172.288,B 90.000,C 0.000} C_DIS
LIN {X 287.368,Y -38.980,Z 178.174,A 172.275,B 90.000,C 0.000} C_DIS
LIN {X 287.363,Y -39.022,Z 178.123,A 172.267,B 90.000,C 0.000} C_DIS
LIN {X 287.335,Y -39.225,Z 178.081,A 172.227,B 90.000,C 0.000} C_DIS
LIN {X 287.329,Y -39.267,Z 178.030,A 172.218,B 90.000,C 0.000} C_DIS
LIN {X 287.321,Y -39.330,Z 177.978,A 172.206,B 90.000,C 0.000} C_DIS
LIN {X 287.279,Y -39.633,Z 177.936,A 172.145,B 90.000,C 0.000} C_DIS
LIN {X 287.262,Y -39.759,Z 177.834,A 172.120,B 90.000,C 0.000} C_DIS
LIN {X 287.219,Y -40.063,Z 177.792,A 172.059,B 90.000,C 0.000} C_DIS
LIN {X 287.202,Y -40.189,Z 177.689,A 172.034,B 90.000,C 0.000} C_DIS
LIN {X 287.159,Y -40.492,Z 177.647,A 171.974,B 90.000,C 0.000} C_DIS
LIN {X 287.150,Y -40.555,Z 177.596,A 171.961,B 90.000,C 0.000} C_DIS
LIN {X 287.144,Y -40.597,Z 177.545,A 171.953,B 90.000,C 0.000} C_DIS
LIN {X 287.116,Y -40.799,Z 177.502,A 171.912,B 90.000,C 0.000} C_DIS
LIN {X 287.110,Y -40.841,Z 177.451,A 171.904,B 90.000,C 0.000} C_DIS
LIN {X 287.101,Y -40.904,Z 177.400,A 171.891,B 90.000,C 0.000} C_DIS
LIN {X 287.057,Y -41.207,Z 177.358,A 171.831,B 90.000,C 0.000} C_DIS
LIN {X 287.039,Y -41.334,Z 177.256,A 171.806,B 90.000,C 0.000} C_DIS
LIN {X 286.995,Y -41.637,Z 177.213,A 171.745,B 90.000,C 0.000} C_DIS
LIN {X 286.977,Y -41.763,Z 177.111,A 171.720,B 90.000,C 0.000} C_DIS
LIN {X 286.933,Y -42.066,Z 177.069,A 171.660,B 90.000,C 0.000} C_DIS
LIN {X 286.924,Y -42.129,Z 177.018,A 171.647,B 90.000,C 0.000} C_DIS
LIN {X 286.917,Y -42.171,Z 176.967,A 171.639,B 90.000,C 0.000} C_DIS
LIN {X 286.888,Y -42.373,Z 176.924,A 171.598,B 90.000,C 0.000} C_DIS
LIN {X 286.882,Y -42.415,Z 176.873,A 171.590,B 90.000,C 0.000} C_DIS
LIN {X 286.872,Y -42.478,Z 176.822,A 171.577,B 90.000,C 0.000} C_DIS
LIN {X 286.827,Y -42.780,Z 176.780,A 171.517,B 90.000,C 0.000} C_DIS
LIN {X 286.808,Y -42.906,Z 176.678,A 171.492,B 90.000,C 0.000} C_DIS
LIN {X 286.763,Y -43.209,Z 176.635,A 171.431,B 90.000,C 0.000} C_DIS
LIN {X 286.753,Y -43.272,Z 176.584,A 171.419,B 90.000,C 0.000} C_DIS
LIN {X 286.747,Y -43.314,Z 176.533,A 171.410,B 90.000,C 0.000} C_DIS
LIN {X 286.716,Y -43.516,Z 176.491,A 171.370,B 90.000,C 0.000} C_DIS
LIN {X 286.710,Y -43.558,Z 176.440,A 171.361,B 90.000,C 0.000} C_DIS
LIN {X 286.701,Y -43.621,Z 176.389,A 171.349,B 90.000,C 0.000} C_DIS
LIN {X 286.654,Y -43.924,Z 176.346,A 171.288,B 90.000,C 0.000} C_DIS
LIN {X 286.635,Y -44.050,Z 176.244,A 171.263,B 90.000,C 0.000} C_DIS
LIN {X 286.588,Y -44.352,Z 176.202,A 171.203,B 90.000,C 0.000} C_DIS
LIN {X 286.569,Y -44.478,Z 176.100,A 171.178,B 90.000,C 0.000} C_DIS
LIN {X 286.522,Y -44.781,Z 176.057,A 171.117,B 90.000,C 0.000} C_DIS
LIN {X 286.512,Y -44.844,Z 176.006,A 171.104,B 90.000,C 0.000} C_DIS
LIN {X 286.505,Y -44.886,Z 175.955,A 171.096,B 90.000,C 0.000} C_DIS
LIN {X 286.474,Y -45.087,Z 175.913,A 171.056,B 90.000,C 0.000} C_DIS
LIN {X 286.467,Y -45.129,Z 175.862,A 171.047,B 90.000,C 0.000} C_DIS
LIN {X 286.457,Y -45.192,Z 175.811,A 171.035,B 90.000,C 0.000} C_DIS
LIN {X 286.409,Y -45.495,Z 175.768,A 170.974,B 90.000,C 0.000} C_DIS
LIN {X 286.389,Y -45.620,Z 175.666,A 170.949,B 90.000,C 0.000} C_DIS
LIN {X 286.341,Y -45.923,Z 175.624,A 170.889,B 90.000,C 0.000} C_DIS
LIN {X 286.321,Y -46.048,Z 175.522,A 170.863,B 90.000,C 0.000} C_DIS
LIN {X 286.272,Y -46.351,Z 175.479,A 170.803,B 90.000,C 0.000} C_DIS
LIN {X 286.262,Y -46.414,Z 175.428,A 170.790,B 90.000,C 0.000} C_DIS
LIN {X 286.255,Y -46.456,Z 175.377,A 170.782,B 90.000,C 0.000} C_DIS
LIN {X 286.222,Y -46.657,Z 175.335,A 170.742,B 90.000,C 0.000} C_DIS
LIN {X 286.215,Y -46.699,Z 175.283,A 170.733,B 90.000,C 0.000} C_DIS
LIN {X 286.205,Y -46.762,Z 175.232,A 170.721,B 90.000,C 0.000} C_DIS
LIN {X 286.156,Y -47.064,Z 175.190,A 170.660,B 90.000,C 0.000} C_DIS
LIN {X 286.135,Y -47.190,Z 175.088,A 170.635,B 90.000,C 0.000} C_DIS
LIN {X 286.085,Y -47.492,Z 175.045,A 170.575,B 90.000,C 0.000} C_DIS
LIN {X 286.074,Y -47.555,Z 174.994,A 170.562,B 90.000,C 0.000} C_DIS
LIN {X 286.067,Y -47.596,Z 174.943,A 170.554,B 90.000,C 0.000} C_DIS
LIN {X 286.034,Y -47.798,Z 174.901,A 170.513,B 90.000,C 0.000} C_DIS
LIN {X 286.027,Y -47.840,Z 174.850,A 170.505,B 90.000,C 0.000} C_DIS
LIN {X 286.016,Y -47.902,Z 174.799,A 170.492,B 90.000,C 0.000} C_DIS
LIN {X 285.966,Y -48.204,Z 174.756,A 170.432,B 90.000,C 0.000} C_DIS
LIN {X 285.944,Y -48.330,Z 174.654,A 170.407,B 90.000,C 0.000} C_DIS
LIN {X 285.893,Y -48.632,Z 174.612,A 170.346,B 90.000,C 0.000} C_DIS
LIN {X 285.872,Y -48.758,Z 174.510,A 170.321,B 90.000,C 0.000} C_DIS
LIN {X 285.820,Y -49.059,Z 174.467,A 170.260,B 90.000,C 0.000} C_DIS
LIN {X 285.809,Y -49.122,Z 174.416,A 170.248,B 90.000,C 0.000} C_DIS
LIN {X 285.802,Y -49.164,Z 174.365,A 170.239,B 90.000,C 0.000} C_DIS
LIN {X 285.768,Y -49.365,Z 174.323,A 170.199,B 90.000,C 0.000} C_DIS
LIN {X 285.760,Y -49.407,Z 174.272,A 170.191,B 90.000,C 0.000} C_DIS
LIN {X 285.749,Y -49.470,Z 174.221,A 170.178,B 90.000,C 0.000} C_DIS
LIN {X 285.697,Y -49.771,Z 174.178,A 170.118,B 90.000,C 0.000} C_DIS
LIN {X 285.675,Y -49.897,Z 174.076,A 170.092,B 90.000,C 0.000} C_DIS
LIN {X 285.622,Y -50.199,Z 174.034,A 170.032,B 90.000,C 0.000} C_DIS
LIN {X 285.600,Y -50.324,Z 173.932,A 170.007,B 90.000,C 0.000} C_DIS
LIN {X 285.547,Y -50.626,Z 173.889,A 169.946,B 90.000,C 0.000} C_DIS
LIN {X 285.536,Y -50.688,Z 173.838,A 169.934,B 90.000,C 0.000} C_DIS
LIN {X 285.528,Y -50.730,Z 173.787,A 169.925,B 90.000,C 0.000} C_DIS
LIN {X 285.493,Y -50.931,Z 173.745,A 169.885,B 90.000,C 0.000} C_DIS
LIN {X 285.485,Y -50.973,Z 173.694,A 169.877,B 90.000,C 0.000} C_DIS
LIN {X 285.474,Y -51.035,Z 173.643,A 169.864,B 90.000,C 0.000} C_DIS
LIN {X 285.420,Y -51.337,Z 173.600,A 169.804,B 90.000,C 0.000} C_DIS
LIN {X 285.397,Y -51.462,Z 173.498,A 169.778,B 90.000,C 0.000} C_DIS
LIN {X 285.343,Y -51.764,Z 173.456,A 169.718,B 90.000,C 0.000} C_DIS
LIN {X 285.331,Y -51.826,Z 173.405,A 169.705,B 90.000,C 0.000} C_DIS
LIN {X 285.324,Y -51.868,Z 173.354,A 169.697,B 90.000,C 0.000} C_DIS
LIN {X 285.287,Y -52.069,Z 173.311,A 169.657,B 90.000,C 0.000} C_DIS
LIN {X 285.280,Y -52.111,Z 173.260,A 169.648,B 90.000,C 0.000} C_DIS
LIN {X 285.268,Y -52.173,Z 173.209,A 169.636,B 90.000,C 0.000} C_DIS
LIN {X 285.213,Y -52.474,Z 173.167,A 169.575,B 90.000,C 0.000} C_DIS
LIN {X 285.190,Y -52.600,Z 173.065,A 169.550,B 90.000,C 0.000} C_DIS
LIN {X 285.134,Y -52.901,Z 173.022,A 169.489,B 90.000,C 0.000} C_DIS
LIN {X 285.111,Y -53.026,Z 172.920,A 169.464,B 90.000,C 0.000} C_DIS
LIN {X 285.055,Y -53.327,Z 172.878,A 169.404,B 90.000,C 0.000} C_DIS
LIN {X 285.043,Y -53.390,Z 172.827,A 169.391,B 90.000,C 0.000} C_DIS
LIN {X 285.035,Y -53.431,Z 172.775,A 169.383,B 90.000,C 0.000} C_DIS
LIN {X 284.998,Y -53.632,Z 172.733,A 169.342,B 90.000,C 0.000} C_DIS
LIN {X 284.990,Y -53.674,Z 172.682,A 169.334,B 90.000,C 0.000} C_DIS
LIN {X 284.978,Y -53.736,Z 172.631,A 169.322,B 90.000,C 0.000} C_DIS
LIN {X 284.921,Y -54.037,Z 172.588,A 169.261,B 90.000,C 0.000} C_DIS
LIN {X 284.897,Y -54.162,Z 172.486,A 169.236,B 90.000,C 0.000} C_DIS
LIN {X 284.840,Y -54.463,Z 172.444,A 169.175,B 90.000,C 0.000} C_DIS
LIN {X 284.816,Y -54.588,Z 172.342,A 169.150,B 90.000,C 0.000} C_DIS
LIN {X 284.758,Y -54.889,Z 172.299,A 169.090,B 90.000,C 0.000} C_DIS
LIN {X 284.746,Y -54.952,Z 172.248,A 169.077,B 90.000,C 0.000} C_DIS
LIN {X 284.738,Y -54.993,Z 172.197,A 169.069,B 90.000,C 0.000} C_DIS
LIN {X 284.699,Y -55.194,Z 172.155,A 169.028,B 90.000,C 0.000} C_DIS
LIN {X 284.691,Y -55.235,Z 172.104,A 169.020,B 90.000,C 0.000} C_DIS
LIN {X 284.679,Y -55.298,Z 172.053,A 169.007,B 90.000,C 0.000} C_DIS
LIN {X 284.620,Y -55.598,Z 172.010,A 168.947,B 90.000,C 0.000} C_DIS
LIN {X 284.596,Y -55.723,Z 171.908,A 168.922,B 90.000,C 0.000} C_DIS
LIN {X 284.537,Y -56.024,Z 171.866,A 168.861,B 90.000,C 0.000} C_DIS
LIN {X 284.525,Y -56.086,Z 171.815,A 168.849,B 90.000,C 0.000} C_DIS
LIN {X 284.517,Y -56.128,Z 171.764,A 168.840,B 90.000,C 0.000} C_DIS
LIN {X 284.477,Y -56.328,Z 171.721,A 168.800,B 90.000,C 0.000} C_DIS
LIN {X 284.469,Y -56.370,Z 171.670,A 168.792,B 90.000,C 0.000} C_DIS
LIN {X 284.456,Y -56.432,Z 171.619,A 168.779,B 90.000,C 0.000} C_DIS
LIN {X 284.397,Y -56.733,Z 171.577,A 168.718,B 90.000,C 0.000} C_DIS
LIN {X 284.372,Y -56.858,Z 171.475,A 168.693,B 90.000,C 0.000} C_DIS
LIN {X 284.311,Y -57.158,Z 171.432,A 168.633,B 90.000,C 0.000} C_DIS
LIN {X 284.286,Y -57.283,Z 171.330,A 168.608,B 90.000,C 0.000} C_DIS
LIN {X 284.226,Y -57.583,Z 171.288,A 168.547,B 90.000,C 0.000} C_DIS
LIN {X 284.213,Y -57.645,Z 171.237,A 168.535,B 90.000,C 0.000} C_DIS
LIN {X 284.205,Y -57.687,Z 171.186,A 168.526,B 90.000,C 0.000} C_DIS
LIN {X 284.164,Y -57.887,Z 171.143,A 168.486,B 90.000,C 0.000} C_DIS
LIN {X 284.155,Y -57.929,Z 171.092,A 168.477,B 90.000,C 0.000} C_DIS
LIN {X 284.143,Y -57.991,Z 171.041,A 168.465,B 90.000,C 0.000} C_DIS
LIN {X 284.081,Y -58.291,Z 170.999,A 168.404,B 90.000,C 0.000} C_DIS
LIN {X 284.056,Y -58.416,Z 170.897,A 168.379,B 90.000,C 0.000} C_DIS
LIN {X 283.994,Y -58.716,Z 170.854,A 168.319,B 90.000,C 0.000} C_DIS
LIN {X 283.968,Y -58.840,Z 170.752,A 168.294,B 90.000,C 0.000} C_DIS
LIN {X 283.906,Y -59.140,Z 170.710,A 168.233,B 90.000,C 0.000} C_DIS
LIN {X 283.893,Y -59.203,Z 170.659,A 168.220,B 90.000,C 0.000} C_DIS
LIN {X 283.884,Y -59.244,Z 170.608,A 168.212,B 90.000,C 0.000} C_DIS
LIN {X 283.842,Y -59.444,Z 170.565,A 168.172,B 90.000,C 0.000} C_DIS
LIN {X 283.834,Y -59.485,Z 170.514,A 168.163,B 90.000,C 0.000} C_DIS
LIN {X 283.820,Y -59.548,Z 170.463,A 168.151,B 90.000,C 0.000} C_DIS
LIN {X 283.757,Y -59.847,Z 170.421,A 168.090,B 90.000,C 0.000} C_DIS
LIN {X 283.731,Y -59.972,Z 170.319,A 168.065,B 90.000,C 0.000} C_DIS
LIN {X 283.668,Y -60.272,Z 170.276,A 168.005,B 90.000,C 0.000} C_DIS
LIN {X 283.654,Y -60.334,Z 170.225,A 167.992,B 90.000,C 0.000} C_DIS
LIN {X 283.646,Y -60.375,Z 170.174,A 167.984,B 90.000,C 0.000} C_DIS
LIN {X 283.603,Y -60.575,Z 170.132,A 167.943,B 90.000,C 0.000} C_DIS
LIN {X 283.594,Y -60.617,Z 170.080,A 167.935,B 90.000,C 0.000} C_DIS
LIN {X 283.581,Y -60.679,Z 170.029,A 167.922,B 90.000,C 0.000} C_DIS
LIN {X 283.517,Y -60.978,Z 169.987,A 167.862,B 90.000,C 0.000} C_DIS
LIN {X 283.490,Y -61.103,Z 169.885,A 167.837,B 90.000,C 0.000} C_DIS
LIN {X 283.425,Y -61.402,Z 169.842,A 167.776,B 90.000,C 0.000} C_DIS
LIN {X 283.398,Y -61.527,Z 169.740,A 167.751,B 90.000,C 0.000} C_DIS
LIN {X 283.333,Y -61.826,Z 169.698,A 167.690,B 90.000,C 0.000} C_DIS
LIN {X 283.319,Y -61.888,Z 169.647,A 167.678,B 90.000,C 0.000} C_DIS
LIN {X 283.310,Y -61.929,Z 169.596,A 167.670,B 90.000,C 0.000} C_DIS
LIN {X 283.267,Y -62.129,Z 169.553,A 167.629,B 90.000,C 0.000} C_DIS
LIN {X 283.258,Y -62.170,Z 169.502,A 167.621,B 90.000,C 0.000} C_DIS
LIN {X 283.244,Y -62.233,Z 169.451,A 167.608,B 90.000,C 0.000} C_DIS
LIN {X 283.178,Y -62.532,Z 169.409,A 167.548,B 90.000,C 0.000} C_DIS
LIN {X 283.151,Y -62.656,Z 169.307,A 167.523,B 90.000,C 0.000} C_DIS
LIN {X 283.084,Y -62.955,Z 169.264,A 167.462,B 90.000,C 0.000} C_DIS
LIN {X 283.070,Y -63.017,Z 169.213,A 167.449,B 90.000,C 0.000} C_DIS
LIN {X 283.061,Y -63.059,Z 169.162,A 167.441,B 90.000,C 0.000} C_DIS
LIN {X 283.017,Y -63.258,Z 169.120,A 167.401,B 90.000,C 0.000} C_DIS
LIN {X 283.007,Y -63.299,Z 169.069,A 167.392,B 90.000,C 0.000} C_DIS
LIN {X 282.994,Y -63.361,Z 169.018,A 167.380,B 90.000,C 0.000} C_DIS
LIN {X 282.926,Y -63.660,Z 168.975,A 167.319,B 90.000,C 0.000} C_DIS
LIN {X 282.898,Y -63.784,Z 168.873,A 167.294,B 90.000,C 0.000} C_DIS
LIN {X 282.831,Y -64.083,Z 168.831,A 167.234,B 90.000,C 0.000} C_DIS
LIN {X 282.803,Y -64.207,Z 168.729,A 167.208,B 90.000,C 0.000} C_DIS
LIN {X 282.735,Y -64.506,Z 168.686,A 167.148,B 90.000,C 0.000} C_DIS
LIN {X 282.721,Y -64.568,Z 168.635,A 167.135,B 90.000,C 0.000} C_DIS
LIN {X 282.711,Y -64.609,Z 168.584,A 167.127,B 90.000,C 0.000} C_DIS
LIN {X 282.666,Y -64.808,Z 168.542,A 167.087,B 90.000,C 0.000} C_DIS
LIN {X 282.656,Y -64.850,Z 168.491,A 167.078,B 90.000,C 0.000} C_DIS
LIN {X 282.642,Y -64.912,Z 168.440,A 167.066,B 90.000,C 0.000} C_DIS
LIN {X 282.573,Y -65.210,Z 168.397,A 167.005,B 90.000,C 0.000} C_DIS
LIN {X 282.545,Y -65.334,Z 168.295,A 166.980,B 90.000,C 0.000} C_DIS
LIN {X 282.475,Y -65.633,Z 168.253,A 166.920,B 90.000,C 0.000} C_DIS
LIN {X 282.447,Y -65.757,Z 168.151,A 166.894,B 90.000,C 0.000} C_DIS
LIN {X 282.377,Y -66.055,Z 168.108,A 166.834,B 90.000,C 0.000} C_DIS
LIN {X 282.362,Y -66.117,Z 168.057,A 166.821,B 90.000,C 0.000} C_DIS
LIN {X 282.353,Y -66.158,Z 168.006,A 166.813,B 90.000,C 0.000} C_DIS
LIN {X 282.306,Y -66.357,Z 167.964,A 166.773,B 90.000,C 0.000} C_DIS
LIN {X 282.296,Y -66.398,Z 167.913,A 166.764,B 90.000,C 0.000} C_DIS
LIN {X 282.282,Y -66.460,Z 167.862,A 166.752,B 90.000,C 0.000} C_DIS
LIN {X 282.211,Y -66.758,Z 167.819,A 166.691,B 90.000,C 0.000} C_DIS
LIN {X 282.182,Y -66.882,Z 167.717,A 166.666,B 90.000,C 0.000} C_DIS
LIN {X 282.111,Y -67.180,Z 167.675,A 166.605,B 90.000,C 0.000} C_DIS
LIN {X 282.082,Y -67.304,Z 167.572,A 166.580,B 90.000,C 0.000} C_DIS
LIN {X 282.011,Y -67.602,Z 167.530,A 166.520,B 90.000,C 0.000} C_DIS
LIN {X 281.996,Y -67.664,Z 167.479,A 166.507,B 90.000,C 0.000} C_DIS
LIN {X 281.986,Y -67.705,Z 167.428,A 166.499,B 90.000,C 0.000} C_DIS
LIN {X 281.938,Y -67.904,Z 167.385,A 166.458,B 90.000,C 0.000} C_DIS
LIN {X 281.928,Y -67.945,Z 167.334,A 166.450,B 90.000,C 0.000} C_DIS
LIN {X 281.913,Y -68.007,Z 167.283,A 166.437,B 90.000,C 0.000} C_DIS
LIN {X 281.841,Y -68.304,Z 167.241,A 166.377,B 90.000,C 0.000} C_DIS
LIN {X 281.811,Y -68.428,Z 167.139,A 166.352,B 90.000,C 0.000} C_DIS
LIN {X 281.739,Y -68.726,Z 167.096,A 166.291,B 90.000,C 0.000} C_DIS
LIN {X 281.724,Y -68.788,Z 167.045,A 166.279,B 90.000,C 0.000} C_DIS
LIN {X 281.714,Y -68.829,Z 166.994,A 166.270,B 90.000,C 0.000} C_DIS
LIN {X 281.665,Y -69.027,Z 166.952,A 166.230,B 90.000,C 0.000} C_DIS
LIN {X 281.655,Y -69.068,Z 166.901,A 166.222,B 90.000,C 0.000} C_DIS
LIN {X 281.640,Y -69.130,Z 166.850,A 166.209,B 90.000,C 0.000} C_DIS
LIN {X 281.567,Y -69.428,Z 166.807,A 166.149,B 90.000,C 0.000} C_DIS
LIN {X 281.536,Y -69.551,Z 166.705,A 166.123,B 90.000,C 0.000} C_DIS
LIN {X 281.463,Y -69.848,Z 166.663,A 166.063,B 90.000,C 0.000} C_DIS
LIN {X 281.432,Y -69.972,Z 166.561,A 166.038,B 90.000,C 0.000} C_DIS
LIN {X 281.358,Y -70.269,Z 166.518,A 165.977,B 90.000,C 0.000} C_DIS
LIN {X 281.342,Y -70.331,Z 166.467,A 165.965,B 90.000,C 0.000} C_DIS
LIN {X 281.332,Y -70.372,Z 166.416,A 165.956,B 90.000,C 0.000} C_DIS
LIN {X 281.282,Y -70.570,Z 166.374,A 165.916,B 90.000,C 0.000} C_DIS
LIN {X 281.272,Y -70.611,Z 166.323,A 165.908,B 90.000,C 0.000} C_DIS
LIN {X 281.257,Y -70.673,Z 166.272,A 165.895,B 90.000,C 0.000} C_DIS
LIN {X 281.182,Y -70.970,Z 166.229,A 165.834,B 90.000,C 0.000} C_DIS
LIN {X 281.151,Y -71.094,Z 166.127,A 165.809,B 90.000,C 0.000} C_DIS
LIN {X 281.075,Y -71.390,Z 166.085,A 165.749,B 90.000,C 0.000} C_DIS
LIN {X 281.060,Y -71.452,Z 166.034,A 165.736,B 90.000,C 0.000} C_DIS
LIN {X 281.049,Y -71.493,Z 165.983,A 165.728,B 90.000,C 0.000} C_DIS
LIN {X 280.999,Y -71.691,Z 165.940,A 165.687,B 90.000,C 0.000} C_DIS
LIN {X 280.988,Y -71.732,Z 165.889,A 165.679,B 90.000,C 0.000} C_DIS
LIN {X 280.973,Y -71.794,Z 165.838,A 165.667,B 90.000,C 0.000} C_DIS
LIN {X 280.897,Y -72.091,Z 165.796,A 165.606,B 90.000,C 0.000} C_DIS
LIN {X 280.865,Y -72.214,Z 165.694,A 165.581,B 90.000,C 0.000} C_DIS
LIN {X 280.789,Y -72.511,Z 165.651,A 165.520,B 90.000,C 0.000} C_DIS
LIN {X 280.757,Y -72.634,Z 165.549,A 165.495,B 90.000,C 0.000} C_DIS
LIN {X 280.680,Y -72.930,Z 165.507,A 165.435,B 90.000,C 0.000} C_DIS
LIN {X 280.664,Y -72.992,Z 165.456,A 165.422,B 90.000,C 0.000} C_DIS
LIN {X 280.653,Y -73.033,Z 165.405,A 165.414,B 90.000,C 0.000} C_DIS
LIN {X 280.602,Y -73.231,Z 165.362,A 165.373,B 90.000,C 0.000} C_DIS
LIN {X 280.591,Y -73.272,Z 165.311,A 165.365,B 90.000,C 0.000} C_DIS
LIN {X 280.575,Y -73.333,Z 165.260,A 165.352,B 90.000,C 0.000} C_DIS
LIN {X 280.497,Y -73.629,Z 165.218,A 165.292,B 90.000,C 0.000} C_DIS
LIN {X 280.465,Y -73.753,Z 165.115,A 165.267,B 90.000,C 0.000} C_DIS
LIN {X 280.387,Y -74.049,Z 165.073,A 165.206,B 90.000,C 0.000} C_DIS
LIN {X 280.354,Y -74.172,Z 164.971,A 165.181,B 90.000,C 0.000} C_DIS
LIN {X 280.276,Y -74.468,Z 164.929,A 165.121,B 90.000,C 0.000} C_DIS
LIN {X 280.259,Y -74.529,Z 164.877,A 165.108,B 90.000,C 0.000} C_DIS
LIN {X 280.249,Y -74.570,Z 164.826,A 165.100,B 90.000,C 0.000} C_DIS
LIN {X 280.196,Y -74.768,Z 164.784,A 165.059,B 90.000,C 0.000} C_DIS
LIN {X 280.185,Y -74.809,Z 164.733,A 165.051,B 90.000,C 0.000} C_DIS
LIN {X 280.169,Y -74.870,Z 164.682,A 165.038,B 90.000,C 0.000} C_DIS
LIN {X 280.089,Y -75.166,Z 164.639,A 164.978,B 90.000,C 0.000} C_DIS
LIN {X 280.057,Y -75.287,Z 164.537,A 164.953,B 90.000,C 0.000} C_DIS
LIN {X 279.977,Y -75.583,Z 164.490,A 164.892,B 90.000,C 0.000} C_DIS
LIN {X 279.956,Y -75.663,Z 164.428,A 164.876,B 90.000,C 0.000} C_DIS
LIN {X 279.905,Y -75.849,Z 164.539,A 164.838,B 90.000,C 0.000} C_DIS
LIN {X 279.639,Y -76.826,Z 165.528,A 164.638,B 90.000,C 0.000} C_DIS
LIN {X 279.013,Y -79.067,Z 165.509,A 164.178,B 90.000,C 0.000} C_DIS
LIN {X 278.838,Y -79.684,Z 165.403,A 164.051,B 90.000,C 0.000} C_DIS
LIN {X 278.397,Y -81.212,Z 165.364,A 163.737,B 90.000,C 0.000} C_DIS
LIN {X 278.229,Y -81.784,Z 165.258,A 163.620,B 90.000,C 0.000} C_DIS
LIN {X 277.745,Y -83.412,Z 165.220,A 163.284,B 90.000,C 0.000} C_DIS
LIN {X 277.568,Y -84.000,Z 165.113,A 163.163,B 90.000,C 0.000} C_DIS
LIN {X 277.071,Y -85.624,Z 165.075,A 162.827,B 90.000,C 0.000} C_DIS
LIN {X 276.889,Y -86.211,Z 164.969,A 162.706,B 90.000,C 0.000} C_DIS
LIN {X 276.380,Y -87.831,Z 164.931,A 162.370,B 90.000,C 0.000} C_DIS
LIN {X 276.201,Y -88.391,Z 164.825,A 162.254,B 90.000,C 0.000} C_DIS
LIN {X 275.678,Y -90.011,Z 164.829,A 161.918,B 90.000,C 0.000} C_DIS
LIN {X 275.623,Y -90.177,Z 164.882,A 161.883,B 90.000,C 0.000} C_DIS
LIN {X 275.585,Y -90.292,Z 164.983,A 161.859,B 90.000,C 0.000} C_DIS
LIN {X 275.499,Y -90.555,Z 165.393,A 161.805,B 90.000,C 0.000} C_DIS
LIN {X 275.352,Y -91.001,Z 165.863,A 161.712,B 90.000,C 0.000} C_DIS
LIN {X 275.303,Y -91.150,Z 165.961,A 161.681,B 90.000,C 0.000} C_DIS
LIN {X 275.080,Y -91.822,Z 166.578,A 161.541,B 90.000,C 0.000} C_DIS
LIN {X 274.961,Y -92.176,Z 166.829,A 161.467,B 90.000,C 0.000} C_DIS
LIN {X 274.927,Y -92.277,Z 166.931,A 161.446,B 90.000,C 0.000} C_DIS
LIN {X 274.857,Y -92.485,Z 167.016,A 161.403,B 90.000,C 0.000} C_DIS
LIN {X 274.788,Y -92.692,Z 167.220,A 161.360,B 90.000,C 0.000} C_DIS
LIN {X 274.749,Y -92.807,Z 167.262,A 161.336,B 90.000,C 0.000} C_DIS
LIN {X 274.720,Y -92.893,Z 167.283,A 161.318,B 90.000,C 0.000} C_DIS
LIN {X 274.694,Y -92.969,Z 167.385,A 161.302,B 90.000,C 0.000} C_DIS
LIN {X 274.628,Y -93.162,Z 167.428,A 161.261,B 90.000,C 0.000} C_DIS
LIN {X 274.601,Y -93.243,Z 167.530,A 161.245,B 90.000,C 0.000} C_DIS
LIN {X 274.535,Y -93.436,Z 167.572,A 161.204,B 90.000,C 0.000} C_DIS
LIN {X 274.508,Y -93.516,Z 167.675,A 161.188,B 90.000,C 0.000} C_DIS
LIN {X 274.442,Y -93.710,Z 167.717,A 161.147,B 90.000,C 0.000} C_DIS
LIN {X 274.428,Y -93.750,Z 167.768,A 161.139,B 90.000,C 0.000} C_DIS
LIN {X 274.408,Y -93.810,Z 167.819,A 161.126,B 90.000,C 0.000} C_DIS
LIN {X 274.309,Y -94.100,Z 167.862,A 161.066,B 90.000,C 0.000} C_DIS
LIN {X 274.288,Y -94.160,Z 167.913,A 161.053,B 90.000,C 0.000} C_DIS
LIN {X 274.274,Y -94.200,Z 167.964,A 161.045,B 90.000,C 0.000} C_DIS
LIN {X 274.208,Y -94.393,Z 168.006,A 161.004,B 90.000,C 0.000} C_DIS
LIN {X 274.194,Y -94.433,Z 168.057,A 160.996,B 90.000,C 0.000} C_DIS
LIN {X 274.166,Y -94.514,Z 168.108,A 160.979,B 90.000,C 0.000} C_DIS
LIN {X 274.033,Y -94.900,Z 168.151,A 160.899,B 90.000,C 0.000} C_DIS
LIN {X 274.005,Y -94.980,Z 168.202,A 160.882,B 90.000,C 0.000} C_DIS
LIN {X 273.984,Y -95.040,Z 168.253,A 160.869,B 90.000,C 0.000} C_DIS
LIN {X 273.884,Y -95.329,Z 168.295,A 160.809,B 90.000,C 0.000} C_DIS
LIN {X 273.863,Y -95.389,Z 168.346,A 160.796,B 90.000,C 0.000} C_DIS
LIN {X 273.821,Y -95.509,Z 168.397,A 160.771,B 90.000,C 0.000} C_DIS
LIN {X 273.618,Y -96.089,Z 168.439,A 160.650,B 90.000,C 0.000} C_DIS
LIN {X 273.576,Y -96.208,Z 168.491,A 160.625,B 90.000,C 0.000} C_DIS
LIN {X 273.444,Y -96.583,Z 168.544,A 160.546,B 90.000,C 0.000} C_DIS
LIN {X 272.690,Y -98.692,Z 168.544,A 160.104,B 90.000,C 0.000} C_DIS
LIN {X 272.555,Y -99.066,Z 168.491,A 160.025,B 90.000,C 0.000} C_DIS
LIN {X 272.518,Y -99.166,Z 168.440,A 160.004,B 90.000,C 0.000} C_DIS
LIN {X 272.343,Y -99.645,Z 168.397,A 159.903,B 90.000,C 0.000} C_DIS
LIN {X 272.278,Y -99.824,Z 168.295,A 159.866,B 90.000,C 0.000} C_DIS
LIN {X 272.137,Y -100.208,Z 168.253,A 159.785,B 90.000,C 0.000} C_DIS
LIN {X 272.107,Y -100.287,Z 168.202,A 159.768,B 90.000,C 0.000} C_DIS
LIN {X 272.085,Y -100.347,Z 168.151,A 159.756,B 90.000,C 0.000} C_DIS
LIN {X 271.979,Y -100.634,Z 168.108,A 159.695,B 90.000,C 0.000} C_DIS
LIN {X 271.935,Y -100.754,Z 168.006,A 159.670,B 90.000,C 0.000} C_DIS
LIN {X 271.829,Y -101.041,Z 167.964,A 159.610,B 90.000,C 0.000} C_DIS
LIN {X 271.806,Y -101.101,Z 167.913,A 159.597,B 90.000,C 0.000} C_DIS
LIN {X 271.792,Y -101.140,Z 167.862,A 159.589,B 90.000,C 0.000} C_DIS
LIN {X 271.720,Y -101.332,Z 167.819,A 159.548,B 90.000,C 0.000} C_DIS
LIN {X 271.691,Y -101.411,Z 167.717,A 159.531,B 90.000,C 0.000} C_DIS
LIN {X 271.619,Y -101.602,Z 167.675,A 159.491,B 90.000,C 0.000} C_DIS
LIN {X 271.589,Y -101.682,Z 167.572,A 159.474,B 90.000,C 0.000} C_DIS
LIN {X 271.518,Y -101.873,Z 167.530,A 159.434,B 90.000,C 0.000} C_DIS
LIN {X 271.488,Y -101.953,Z 167.428,A 159.417,B 90.000,C 0.000} C_DIS
LIN {X 271.416,Y -102.144,Z 167.385,A 159.377,B 90.000,C 0.000} C_DIS
LIN {X 271.386,Y -102.223,Z 167.283,A 159.360,B 90.000,C 0.000} C_DIS
LIN {X 271.314,Y -102.414,Z 167.241,A 159.320,B 90.000,C 0.000} C_DIS
LIN {X 271.286,Y -102.489,Z 167.139,A 159.304,B 90.000,C 0.000} C_DIS
LIN {X 271.254,Y -102.574,Z 167.118,A 159.286,B 90.000,C 0.000} C_DIS
LIN {X 271.211,Y -102.688,Z 167.075,A 159.262,B 90.000,C 0.000} C_DIS
LIN {X 271.135,Y -102.888,Z 166.871,A 159.220,B 90.000,C 0.000} C_DIS
LIN {X 271.053,Y -103.104,Z 166.765,A 159.174,B 90.000,C 0.000} C_DIS
LIN {X 270.395,Y -104.818,Z 165.068,A 158.811,B 90.000,C 0.000} C_DIS
LIN {X 270.183,Y -105.363,Z 164.344,A 158.696,B 90.000,C 0.000} C_DIS
LIN {X 270.144,Y -105.462,Z 164.113,A 158.675,B 90.000,C 0.000} C_DIS
LIN {X 270.070,Y -105.652,Z 163.899,A 158.634,B 90.000,C 0.000} C_DIS
LIN {X 270.054,Y -105.691,Z 163.778,A 158.626,B 90.000,C 0.000} C_DIS
LIN {X 270.047,Y -105.711,Z 163.687,A 158.622,B 90.000,C 0.000} C_DIS
LIN {X 270.009,Y -105.806,Z 163.607,A 158.602,B 90.000,C 0.000} C_DIS
LIN {X 269.994,Y -105.846,Z 163.402,A 158.593,B 90.000,C 0.000} C_DIS
LIN {X 269.957,Y -105.941,Z 163.317,A 158.573,B 90.000,C 0.000} C_DIS
LIN {X 269.941,Y -105.980,Z 163.113,A 158.565,B 90.000,C 0.000} C_DIS
LIN {X 269.904,Y -106.075,Z 163.028,A 158.545,B 90.000,C 0.000} C_DIS
LIN {X 269.888,Y -106.115,Z 162.824,A 158.536,B 90.000,C 0.000} C_DIS
LIN {X 269.851,Y -106.210,Z 162.739,A 158.516,B 90.000,C 0.000} C_DIS
LIN {X 269.835,Y -106.249,Z 162.535,A 158.508,B 90.000,C 0.000} C_DIS
LIN {X 269.798,Y -106.344,Z 162.450,A 158.487,B 90.000,C 0.000} C_DIS
LIN {X 269.782,Y -106.384,Z 162.246,A 158.479,B 90.000,C 0.000} C_DIS
LIN {X 269.764,Y -106.431,Z 162.204,A 158.469,B 90.000,C 0.000} C_DIS
LIN {X 269.745,Y -106.479,Z 162.140,A 158.459,B 90.000,C 0.000} C_DIS
LIN {X 269.729,Y -106.518,Z 161.834,A 158.451,B 90.000,C 0.000} C_DIS
LIN {X 269.692,Y -106.613,Z 161.706,A 158.430,B 90.000,C 0.000} C_DIS
LIN {X 269.676,Y -106.653,Z 161.400,A 158.422,B 90.000,C 0.000} C_DIS
LIN {X 269.657,Y -106.700,Z 161.337,A 158.412,B 90.000,C 0.000} C_DIS
LIN {X 269.639,Y -106.748,Z 161.252,A 158.402,B 90.000,C 0.000} C_DIS
LIN {X 269.623,Y -106.787,Z 160.843,A 158.393,B 90.000,C 0.000} C_DIS
LIN {X 269.585,Y -106.882,Z 160.652,A 158.373,B 90.000,C 0.000} C_DIS
LIN {X 269.570,Y -106.921,Z 160.142,A 158.365,B 90.000,C 0.000} C_DIS
LIN {X 269.551,Y -106.969,Z 160.036,A 158.355,B 90.000,C 0.000} C_DIS
LIN {X 269.531,Y -107.018,Z 159.638,A 158.344,B 90.000,C 0.000} C_DIS
LIN {X 269.531,Y -107.018,Z 157.398,A 158.344,B 90.000,C 0.000} C_DIS
LIN {X 269.551,Y -106.969,Z 157.001,A 158.355,B 90.000,C 0.000} C_DIS
LIN {X 269.570,Y -106.921,Z 156.895,A 158.365,B 90.000,C 0.000} C_DIS
LIN {X 269.585,Y -106.882,Z 156.384,A 158.373,B 90.000,C 0.000} C_DIS
LIN {X 269.623,Y -106.787,Z 156.193,A 158.393,B 90.000,C 0.000} C_DIS
LIN {X 269.639,Y -106.748,Z 155.785,A 158.402,B 90.000,C 0.000} C_DIS
LIN {X 269.657,Y -106.700,Z 155.700,A 158.412,B 90.000,C 0.000} C_DIS
LIN {X 269.676,Y -106.653,Z 155.636,A 158.422,B 90.000,C 0.000} C_DIS
LIN {X 269.692,Y -106.613,Z 155.330,A 158.430,B 90.000,C 0.000} C_DIS
LIN {X 269.729,Y -106.518,Z 155.203,A 158.451,B 90.000,C 0.000} C_DIS
LIN {X 269.745,Y -106.479,Z 154.896,A 158.459,B 90.000,C 0.000} C_DIS
LIN {X 269.782,Y -106.384,Z 154.769,A 158.479,B 90.000,C 0.000} C_DIS
LIN {X 269.798,Y -106.344,Z 154.463,A 158.487,B 90.000,C 0.000} C_DIS
LIN {X 269.817,Y -106.297,Z 154.399,A 158.498,B 90.000,C 0.000} C_DIS
LIN {X 269.835,Y -106.249,Z 154.357,A 158.508,B 90.000,C 0.000} C_DIS
LIN {X 269.851,Y -106.210,Z 154.153,A 158.516,B 90.000,C 0.000} C_DIS
LIN {X 269.888,Y -106.115,Z 154.068,A 158.536,B 90.000,C 0.000} C_DIS
LIN {X 269.904,Y -106.075,Z 153.864,A 158.545,B 90.000,C 0.000} C_DIS
LIN {X 269.941,Y -105.980,Z 153.783,A 158.565,B 90.000,C 0.000} C_DIS
LIN {X 269.949,Y -105.961,Z 153.692,A 158.569,B 90.000,C 0.000} C_DIS
LIN {X 269.964,Y -105.921,Z 153.571,A 158.577,B 90.000,C 0.000} C_DIS
LIN {X 270.039,Y -105.731,Z 153.348,A 158.618,B 90.000,C 0.000} C_DIS
LIN {X 270.054,Y -105.691,Z 153.227,A 158.626,B 90.000,C 0.000} C_DIS
LIN {X 270.062,Y -105.672,Z 153.136,A 158.630,B 90.000,C 0.000} C_DIS
LIN {X 270.099,Y -105.577,Z 153.056,A 158.650,B 90.000,C 0.000} C_DIS
LIN {X 270.107,Y -105.557,Z 152.954,A 158.655,B 90.000,C 0.000} C_DIS
LIN {X 270.090,Y -105.599,Z 152.839,A 158.646,B 90.000,C 0.000} C_DIS
LIN {X 269.972,Y -105.901,Z 152.788,A 158.582,B 90.000,C 0.000} C_DIS
LIN {X 269.949,Y -105.961,Z 152.737,A 158.569,B 90.000,C 0.000} C_DIS
LIN {X 269.933,Y -106.000,Z 152.686,A 158.561,B 90.000,C 0.000} C_DIS
LIN {X 269.859,Y -106.190,Z 152.644,A 158.520,B 90.000,C 0.000} C_DIS
LIN {X 269.843,Y -106.230,Z 152.593,A 158.512,B 90.000,C 0.000} C_DIS
LIN {X 269.820,Y -106.289,Z 152.542,A 158.499,B 90.000,C 0.000} C_DIS
LIN {X 269.707,Y -106.574,Z 152.499,A 158.439,B 90.000,C 0.000} C_DIS
LIN {X 269.661,Y -106.692,Z 152.397,A 158.414,B 90.000,C 0.000} C_DIS
LIN {X 269.548,Y -106.977,Z 152.355,A 158.353,B 90.000,C 0.000} C_DIS
LIN {X 269.501,Y -107.095,Z 152.252,A 158.328,B 90.000,C 0.000} C_DIS
LIN {X 269.387,Y -107.380,Z 152.210,A 158.267,B 90.000,C 0.000} C_DIS
LIN {X 269.364,Y -107.439,Z 152.159,A 158.255,B 90.000,C 0.000} C_DIS
LIN {X 269.348,Y -107.478,Z 152.108,A 158.246,B 90.000,C 0.000} C_DIS
LIN {X 269.310,Y -107.573,Z 152.087,A 158.226,B 90.000,C 0.000} C_DIS
LIN {X 269.282,Y -107.643,Z 152.099,A 158.211,B 90.000,C 0.000} C_DIS
LIN {X 269.266,Y -107.684,Z 152.150,A 158.203,B 90.000,C 0.000} C_DIS
LIN {X 269.249,Y -107.727,Z 152.703,A 158.194,B 90.000,C 0.000} C_DIS
LIN {X 269.211,Y -107.822,Z 152.894,A 158.173,B 90.000,C 0.000} C_DIS
LIN {X 269.195,Y -107.861,Z 153.303,A 158.165,B 90.000,C 0.000} C_DIS
LIN {X 269.157,Y -107.956,Z 153.494,A 158.145,B 90.000,C 0.000} C_DIS
LIN {X 269.141,Y -107.995,Z 154.004,A 158.136,B 90.000,C 0.000} C_DIS
LIN {X 269.103,Y -108.090,Z 154.216,A 158.116,B 90.000,C 0.000} C_DIS
LIN {X 269.087,Y -108.129,Z 154.727,A 158.108,B 90.000,C 0.000} C_DIS
LIN {X 269.049,Y -108.224,Z 154.959,A 158.088,B 90.000,C 0.000} C_DIS
LIN {X 269.034,Y -108.263,Z 155.573,A 158.079,B 90.000,C 0.000} C_DIS
LIN {X 268.995,Y -108.358,Z 155.806,A 158.059,B 90.000,C 0.000} C_DIS
LIN {X 268.979,Y -108.398,Z 156.316,A 158.051,B 90.000,C 0.000} C_DIS
LIN {X 268.941,Y -108.492,Z 156.529,A 158.031,B 90.000,C 0.000} C_DIS
LIN {X 268.925,Y -108.532,Z 157.039,A 158.022,B 90.000,C 0.000} C_DIS
LIN {X 268.887,Y -108.626,Z 157.272,A 158.002,B 90.000,C 0.000} C_DIS
LIN {X 268.871,Y -108.666,Z 157.886,A 157.994,B 90.000,C 0.000} C_DIS
LIN {X 268.833,Y -108.760,Z 158.118,A 157.973,B 90.000,C 0.000} C_DIS
LIN {X 268.817,Y -108.800,Z 158.629,A 157.965,B 90.000,C 0.000} C_DIS
LIN {X 268.779,Y -108.894,Z 158.841,A 157.945,B 90.000,C 0.000} C_DIS
LIN {X 268.763,Y -108.934,Z 159.352,A 157.937,B 90.000,C 0.000} C_DIS
LIN {X 268.724,Y -109.028,Z 159.584,A 157.916,B 90.000,C 0.000} C_DIS
LIN {X 268.709,Y -109.067,Z 160.198,A 157.908,B 90.000,C 0.000} C_DIS
LIN {X 268.689,Y -109.115,Z 160.325,A 157.898,B 90.000,C 0.000} C_DIS
LIN {X 268.670,Y -109.162,Z 160.410,A 157.888,B 90.000,C 0.000} C_DIS
LIN {X 268.654,Y -109.201,Z 160.818,A 157.879,B 90.000,C 0.000} C_DIS
LIN {X 268.635,Y -109.249,Z 160.903,A 157.869,B 90.000,C 0.000} C_DIS
LIN {X 268.616,Y -109.296,Z 160.936,A 157.859,B 90.000,C 0.000} C_DIS
LIN {X 268.608,Y -109.316,Z 161.015,A 157.855,B 90.000,C 0.000} C_DIS
LIN {X 268.588,Y -109.363,Z 161.142,A 157.845,B 90.000,C 0.000} C_DIS
LIN {X 268.543,Y -109.476,Z 161.296,A 157.821,B 90.000,C 0.000} C_DIS
LIN {X 268.488,Y -109.609,Z 161.426,A 157.792,B 90.000,C 0.000} C_DIS
LIN {X 268.443,Y -109.719,Z 161.481,A 157.769,B 90.000,C 0.000} C_DIS
LIN {X 267.704,Y -111.510,Z 163.061,A 157.386,B 90.000,C 0.000} C_DIS
LIN {X 266.948,Y -113.307,Z 164.626,A 157.001,B 90.000,C 0.000} C_DIS
LIN {X 266.261,Y -114.914,Z 166.034,A 156.656,B 90.000,C 0.000} C_DIS
LIN {X 266.181,Y -115.100,Z 166.250,A 156.616,B 90.000,C 0.000} C_DIS
LIN {X 265.178,Y -117.390,Z 166.250,A 156.122,B 90.000,C 0.000} C_DIS
LIN {X 264.157,Y -119.671,Z 166.250,A 155.628,B 90.000,C 0.000} C_DIS
LIN {X 263.115,Y -121.944,Z 166.250,A 155.134,B 90.000,C 0.000} C_DIS
LIN {X 262.054,Y -124.208,Z 166.250,A 154.640,B 90.000,C 0.000} C_DIS
LIN {X 260.974,Y -126.462,Z 166.250,A 154.146,B 90.000,C 0.000} C_DIS
LIN {X 259.874,Y -128.707,Z 166.250,A 153.652,B 90.000,C 0.000} C_DIS
LIN {X 258.755,Y -130.943,Z 166.250,A 153.158,B 90.000,C 0.000} C_DIS
LIN {X 257.616,Y -133.168,Z 166.250,A 152.664,B 90.000,C 0.000} C_DIS
LIN {X 256.459,Y -135.384,Z 166.250,A 152.171,B 90.000,C 0.000} C_DIS
LIN {X 255.883,Y -136.470,Z 166.250,A 151.928,B 90.000,C 0.000} C_DIS
LIN {X 255.752,Y -136.715,Z 165.961,A 151.873,B 90.000,C 0.000} C_DIS
LIN {X 254.827,Y -138.431,Z 164.397,A 151.488,B 90.000,C 0.000} C_DIS
LIN {X 253.895,Y -140.133,Z 162.820,A 151.104,B 90.000,C 0.000} C_DIS
LIN {X 253.012,Y -141.722,Z 161.337,A 150.745,B 90.000,C 0.000} C_DIS
LIN {X 252.919,Y -141.888,Z 161.226,A 150.708,B 90.000,C 0.000} C_DIS
LIN {X 252.870,Y -141.975,Z 161.016,A 150.688,B 90.000,C 0.000} C_DIS
LIN {X 252.860,Y -141.993,Z 160.936,A 150.684,B 90.000,C 0.000} C_DIS
LIN {X 252.835,Y -142.038,Z 160.903,A 150.674,B 90.000,C 0.000} C_DIS
LIN {X 252.810,Y -142.082,Z 160.797,A 150.663,B 90.000,C 0.000} C_DIS
LIN {X 252.789,Y -142.119,Z 160.286,A 150.655,B 90.000,C 0.000} C_DIS
LIN {X 252.739,Y -142.208,Z 160.054,A 150.635,B 90.000,C 0.000} C_DIS
LIN {X 252.718,Y -142.245,Z 159.440,A 150.627,B 90.000,C 0.000} C_DIS
LIN {X 252.668,Y -142.334,Z 159.207,A 150.606,B 90.000,C 0.000} C_DIS
LIN {X 252.647,Y -142.371,Z 158.697,A 150.598,B 90.000,C 0.000} C_DIS
LIN {X 252.597,Y -142.460,Z 158.484,A 150.578,B 90.000,C 0.000} C_DIS
LIN {X 252.576,Y -142.497,Z 157.974,A 150.569,B 90.000,C 0.000} C_DIS
LIN {X 252.526,Y -142.586,Z 157.762,A 150.549,B 90.000,C 0.000} C_DIS
LIN {X 252.505,Y -142.623,Z 157.251,A 150.541,B 90.000,C 0.000} C_DIS
LIN {X 252.455,Y -142.712,Z 157.039,A 150.521,B 90.000,C 0.000} C_DIS
LIN {X 252.434,Y -142.749,Z 156.529,A 150.512,B 90.000,C 0.000} C_DIS
LIN {X 252.384,Y -142.837,Z 156.316,A 150.492,B 90.000,C 0.000} C_DIS
LIN {X 252.363,Y -142.874,Z 155.806,A 150.484,B 90.000,C 0.000} C_DIS
LIN {X 252.312,Y -142.963,Z 155.594,A 150.464,B 90.000,C 0.000} C_DIS
LIN {X 252.291,Y -143.000,Z 155.083,A 150.455,B 90.000,C 0.000} C_DIS
LIN {X 252.241,Y -143.089,Z 154.871,A 150.435,B 90.000,C 0.000} C_DIS
LIN {X 252.220,Y -143.126,Z 154.361,A 150.427,B 90.000,C 0.000} C_DIS
LIN {X 252.170,Y -143.215,Z 154.149,A 150.406,B 90.000,C 0.000} C_DIS
LIN {X 252.149,Y -143.251,Z 153.638,A 150.398,B 90.000,C 0.000} C_DIS
LIN {X 252.098,Y -143.340,Z 153.426,A 150.378,B 90.000,C 0.000} C_DIS
LIN {X 252.077,Y -143.377,Z 152.916,A 150.370,B 90.000,C 0.000} C_DIS
LIN {X 252.052,Y -143.421,Z 152.809,A 150.359,B 90.000,C 0.000} C_DIS
LIN {X 252.027,Y -143.466,Z 152.767,A 150.349,B 90.000,C 0.000} C_DIS
LIN {X 252.016,Y -143.484,Z 152.665,A 150.345,B 90.000,C 0.000} C_DIS
LIN {X 251.999,Y -143.516,Z 152.556,A 150.338,B 90.000,C 0.000} C_DIS
LIN {X 251.945,Y -143.610,Z 152.520,A 150.317,B 90.000,C 0.000} C_DIS
LIN {X 251.894,Y -143.699,Z 152.542,A 150.296,B 90.000,C 0.000} C_DIS
LIN {X 251.873,Y -143.735,Z 152.593,A 150.288,B 90.000,C 0.000} C_DIS
LIN {X 251.842,Y -143.791,Z 152.644,A 150.275,B 90.000,C 0.000} C_DIS
LIN {X 251.690,Y -144.057,Z 152.686,A 150.215,B 90.000,C 0.000} C_DIS
LIN {X 251.626,Y -144.167,Z 152.788,A 150.190,B 90.000,C 0.000} C_DIS
LIN {X 251.474,Y -144.433,Z 152.831,A 150.129,B 90.000,C 0.000} C_DIS
LIN {X 251.442,Y -144.488,Z 152.882,A 150.117,B 90.000,C 0.000} C_DIS
LIN {X 251.421,Y -144.525,Z 152.933,A 150.108,B 90.000,C 0.000} C_DIS
LIN {X 251.319,Y -144.702,Z 152.975,A 150.068,B 90.000,C 0.000} C_DIS
LIN {X 251.298,Y -144.738,Z 153.026,A 150.060,B 90.000,C 0.000} C_DIS
LIN {X 251.266,Y -144.794,Z 153.077,A 150.047,B 90.000,C 0.000} C_DIS
LIN {X 251.113,Y -145.059,Z 153.120,A 149.987,B 90.000,C 0.000} C_DIS
LIN {X 251.081,Y -145.114,Z 153.171,A 149.974,B 90.000,C 0.000} C_DIS
LIN {X 251.060,Y -145.151,Z 153.222,A 149.966,B 90.000,C 0.000} C_DIS
LIN {X 250.957,Y -145.329,Z 153.258,A 149.925,B 90.000,C 0.000} C_DIS
LIN {X 250.940,Y -145.359,Z 153.302,A 149.918,B 90.000,C 0.000} C_DIS
LIN {X 251.060,Y -145.151,Z 153.571,A 149.966,B 90.000,C 0.000} C_DIS
LIN {X 251.081,Y -145.114,Z 153.692,A 149.974,B 90.000,C 0.000} C_DIS
LIN {X 251.092,Y -145.096,Z 153.783,A 149.978,B 90.000,C 0.000} C_DIS
LIN {X 251.143,Y -145.007,Z 153.864,A 149.998,B 90.000,C 0.000} C_DIS
LIN {X 251.164,Y -144.971,Z 154.068,A 150.007,B 90.000,C 0.000} C_DIS
LIN {X 251.215,Y -144.882,Z 154.153,A 150.027,B 90.000,C 0.000} C_DIS
LIN {X 251.237,Y -144.845,Z 154.357,A 150.035,B 90.000,C 0.000} C_DIS
LIN {X 251.262,Y -144.801,Z 154.399,A 150.045,B 90.000,C 0.000} C_DIS
LIN {X 251.288,Y -144.757,Z 154.463,A 150.055,B 90.000,C 0.000} C_DIS
LIN {X 251.309,Y -144.720,Z 154.769,A 150.064,B 90.000,C 0.000} C_DIS
LIN {X 251.360,Y -144.632,Z 154.896,A 150.084,B 90.000,C 0.000} C_DIS
LIN {X 251.381,Y -144.595,Z 155.203,A 150.092,B 90.000,C 0.000} C_DIS
LIN {X 251.432,Y -144.506,Z 155.330,A 150.113,B 90.000,C 0.000} C_DIS
LIN {X 251.453,Y -144.470,Z 155.636,A 150.121,B 90.000,C 0.000} C_DIS
LIN {X 251.478,Y -144.425,Z 155.700,A 150.131,B 90.000,C 0.000} C_DIS
LIN {X 251.504,Y -144.381,Z 155.785,A 150.141,B 90.000,C 0.000} C_DIS
LIN {X 251.525,Y -144.344,Z 156.193,A 150.149,B 90.000,C 0.000} C_DIS
LIN {X 251.576,Y -144.256,Z 156.384,A 150.170,B 90.000,C 0.000} C_DIS
LIN {X 251.597,Y -144.219,Z 156.895,A 150.178,B 90.000,C 0.000} C_DIS
LIN {X 251.622,Y -144.175,Z 157.001,A 150.188,B 90.000,C 0.000} C_DIS
LIN {X 251.649,Y -144.128,Z 157.398,A 150.199,B 90.000,C 0.000} C_DIS
LIN {X 251.649,Y -144.128,Z 159.638,A 150.199,B 90.000,C 0.000} C_DIS
LIN {X 251.622,Y -144.175,Z 160.036,A 150.188,B 90.000,C 0.000} C_DIS
LIN {X 251.597,Y -144.219,Z 160.142,A 150.178,B 90.000,C 0.000} C_DIS
LIN {X 251.576,Y -144.256,Z 160.652,A 150.170,B 90.000,C 0.000} C_DIS
LIN {X 251.525,Y -144.344,Z 160.843,A 150.149,B 90.000,C 0.000} C_DIS
LIN {X 251.504,Y -144.381,Z 161.252,A 150.141,B 90.000,C 0.000} C_DIS
LIN {X 251.478,Y -144.425,Z 161.337,A 150.131,B 90.000,C 0.000} C_DIS
LIN {X 251.453,Y -144.470,Z 161.400,A 150.121,B 90.000,C 0.000} C_DIS
LIN {X 251.432,Y -144.506,Z 161.706,A 150.113,B 90.000,C 0.000} C_DIS
LIN {X 251.381,Y -144.595,Z 161.834,A 150.092,B 90.000,C 0.000} C_DIS
LIN {X 251.360,Y -144.632,Z 162.140,A 150.084,B 90.000,C 0.000} C_DIS
LIN {X 251.334,Y -144.676,Z 162.204,A 150.074,B 90.000,C 0.000} C_DIS
LIN {X 251.309,Y -144.720,Z 162.246,A 150.064,B 90.000,C 0.000} C_DIS
LIN {X 251.288,Y -144.757,Z 162.450,A 150.055,B 90.000,C 0.000} C_DIS
LIN {X 251.237,Y -144.845,Z 162.535,A 150.035,B 90.000,C 0.000} C_DIS
LIN {X 251.215,Y -144.882,Z 162.739,A 150.027,B 90.000,C 0.000} C_DIS
LIN {X 251.164,Y -144.971,Z 162.824,A 150.007,B 90.000,C 0.000} C_DIS
LIN {X 251.143,Y -145.007,Z 163.028,A 149.998,B 90.000,C 0.000} C_DIS
LIN {X 251.092,Y -145.096,Z 163.113,A 149.978,B 90.000,C 0.000} C_DIS
LIN {X 251.071,Y -145.132,Z 163.317,A 149.970,B 90.000,C 0.000} C_DIS
LIN {X 251.020,Y -145.221,Z 163.402,A 149.950,B 90.000,C 0.000} C_DIS
LIN {X 250.998,Y -145.258,Z 163.607,A 149.941,B 90.000,C 0.000} C_DIS
LIN {X 250.947,Y -145.346,Z 163.687,A 149.921,B 90.000,C 0.000} C_DIS
LIN {X 250.937,Y -145.364,Z 163.778,A 149.917,B 90.000,C 0.000} C_DIS
LIN {X 250.915,Y -145.401,Z 163.899,A 149.908,B 90.000,C 0.000} C_DIS
LIN {X 250.813,Y -145.578,Z 164.113,A 149.868,B 90.000,C 0.000} C_DIS
LIN {X 250.760,Y -145.669,Z 164.344,A 149.847,B 90.000,C 0.000} C_DIS
LIN {X 249.903,Y -147.134,Z 166.180,A 149.512,B 90.000,C 0.000} C_DIS
LIN {X 249.535,Y -147.758,Z 166.765,A 149.369,B 90.000,C 0.000} C_DIS
LIN {X 249.417,Y -147.956,Z 166.871,A 149.323,B 90.000,C 0.000} C_DIS
LIN {X 249.308,Y -148.140,Z 167.075,A 149.281,B 90.000,C 0.000} C_DIS
LIN {X 249.246,Y -148.245,Z 167.118,A 149.257,B 90.000,C 0.000} C_DIS
LIN {X 249.199,Y -148.323,Z 167.139,A 149.239,B 90.000,C 0.000} C_DIS
LIN {X 249.158,Y -148.392,Z 167.241,A 149.223,B 90.000,C 0.000} C_DIS
LIN {X 249.054,Y -148.567,Z 167.283,A 149.183,B 90.000,C 0.000} C_DIS
LIN {X 249.010,Y -148.640,Z 167.385,A 149.166,B 90.000,C 0.000} C_DIS
LIN {X 248.906,Y -148.815,Z 167.428,A 149.126,B 90.000,C 0.000} C_DIS
LIN {X 248.862,Y -148.888,Z 167.530,A 149.109,B 90.000,C 0.000} C_DIS
LIN {X 248.757,Y -149.063,Z 167.572,A 149.069,B 90.000,C 0.000} C_DIS
LIN {X 248.714,Y -149.136,Z 167.675,A 149.052,B 90.000,C 0.000} C_DIS
LIN {X 248.609,Y -149.311,Z 167.717,A 149.012,B 90.000,C 0.000} C_DIS
LIN {X 248.565,Y -149.384,Z 167.819,A 148.995,B 90.000,C 0.000} C_DIS
LIN {X 248.460,Y -149.559,Z 167.862,A 148.954,B 90.000,C 0.000} C_DIS
LIN {X 248.438,Y -149.595,Z 167.913,A 148.946,B 90.000,C 0.000} C_DIS
LIN {X 248.405,Y -149.650,Z 167.964,A 148.933,B 90.000,C 0.000} C_DIS
LIN {X 248.247,Y -149.912,Z 168.006,A 148.873,B 90.000,C 0.000} C_DIS
LIN {X 248.181,Y -150.021,Z 168.108,A 148.848,B 90.000,C 0.000} C_DIS
LIN {X 248.022,Y -150.283,Z 168.151,A 148.787,B 90.000,C 0.000} C_DIS
LIN {X 247.989,Y -150.337,Z 168.202,A 148.775,B 90.000,C 0.000} C_DIS
LIN {X 247.945,Y -150.410,Z 168.253,A 148.758,B 90.000,C 0.000} C_DIS
LIN {X 247.733,Y -150.759,Z 168.295,A 148.677,B 90.000,C 0.000} C_DIS
LIN {X 247.634,Y -150.922,Z 168.397,A 148.639,B 90.000,C 0.000} C_DIS
LIN {X 247.368,Y -151.358,Z 168.440,A 148.539,B 90.000,C 0.000} C_DIS
LIN {X 247.312,Y -151.448,Z 168.491,A 148.518,B 90.000,C 0.000} C_DIS
LIN {X 247.105,Y -151.787,Z 168.544,A 148.439,B 90.000,C 0.000} C_DIS
LIN {X 245.925,Y -153.691,Z 168.544,A 147.997,B 90.000,C 0.000} C_DIS
LIN {X 245.714,Y -154.028,Z 168.491,A 147.918,B 90.000,C 0.000} C_DIS
LIN {X 245.647,Y -154.135,Z 168.439,A 147.893,B 90.000,C 0.000} C_DIS
LIN {X 245.320,Y -154.655,Z 168.397,A 147.772,B 90.000,C 0.000} C_DIS
LIN {X 245.252,Y -154.762,Z 168.346,A 147.747,B 90.000,C 0.000} C_DIS
LIN {X 245.218,Y -154.816,Z 168.295,A 147.734,B 90.000,C 0.000} C_DIS
LIN {X 245.055,Y -155.075,Z 168.253,A 147.674,B 90.000,C 0.000} C_DIS
LIN {X 245.021,Y -155.129,Z 168.202,A 147.661,B 90.000,C 0.000} C_DIS
LIN {X 244.975,Y -155.201,Z 168.151,A 147.644,B 90.000,C 0.000} C_DIS
LIN {X 244.756,Y -155.545,Z 168.108,A 147.564,B 90.000,C 0.000} C_DIS
LIN {X 244.711,Y -155.617,Z 168.057,A 147.547,B 90.000,C 0.000} C_DIS
LIN {X 244.688,Y -155.653,Z 168.006,A 147.538,B 90.000,C 0.000} C_DIS
LIN {X 244.578,Y -155.825,Z 167.964,A 147.498,B 90.000,C 0.000} C_DIS
LIN {X 244.556,Y -155.861,Z 167.913,A 147.490,B 90.000,C 0.000} C_DIS
LIN {X 244.521,Y -155.914,Z 167.862,A 147.477,B 90.000,C 0.000} C_DIS
LIN {X 244.357,Y -156.173,Z 167.819,A 147.417,B 90.000,C 0.000} C_DIS
LIN {X 244.322,Y -156.226,Z 167.768,A 147.404,B 90.000,C 0.000} C_DIS
LIN {X 244.299,Y -156.262,Z 167.717,A 147.396,B 90.000,C 0.000} C_DIS
LIN {X 244.189,Y -156.434,Z 167.675,A 147.355,B 90.000,C 0.000} C_DIS
LIN {X 244.144,Y -156.505,Z 167.572,A 147.339,B 90.000,C 0.000} C_DIS
LIN {X 244.033,Y -156.677,Z 167.530,A 147.298,B 90.000,C 0.000} C_DIS
LIN {X 243.987,Y -156.749,Z 167.428,A 147.281,B 90.000,C 0.000} C_DIS
LIN {X 243.877,Y -156.920,Z 167.385,A 147.241,B 90.000,C 0.000} C_DIS
LIN {X 243.834,Y -156.988,Z 167.283,A 147.225,B 90.000,C 0.000} C_DIS
LIN {X 243.784,Y -157.064,Z 167.262,A 147.207,B 90.000,C 0.000} C_DIS
LIN {X 243.719,Y -157.166,Z 167.220,A 147.183,B 90.000,C 0.000} C_DIS
LIN {X 243.600,Y -157.349,Z 167.016,A 147.140,B 90.000,C 0.000} C_DIS
LIN {X 243.481,Y -157.534,Z 166.931,A 147.097,B 90.000,C 0.000} C_DIS
LIN {X 243.423,Y -157.624,Z 166.829,A 147.076,B 90.000,C 0.000} C_DIS
LIN {X 243.220,Y -157.937,Z 166.578,A 147.002,B 90.000,C 0.000} C_DIS
LIN {X 242.834,Y -158.530,Z 165.961,A 146.862,B 90.000,C 0.000} C_DIS
LIN {X 242.748,Y -158.661,Z 165.863,A 146.831,B 90.000,C 0.000} C_DIS
LIN {X 242.491,Y -159.055,Z 165.393,A 146.738,B 90.000,C 0.000} C_DIS
LIN {X 242.339,Y -159.286,Z 164.983,A 146.684,B 90.000,C 0.000} C_DIS
LIN {X 242.272,Y -159.387,Z 164.882,A 146.660,B 90.000,C 0.000} C_DIS
LIN {X 242.176,Y -159.533,Z 164.829,A 146.625,B 90.000,C 0.000} C_DIS
LIN {X 241.235,Y -160.952,Z 164.825,A 146.289,B 90.000,C 0.000} C_DIS
LIN {X 240.908,Y -161.441,Z 164.931,A 146.173,B 90.000,C 0.000} C_DIS
LIN {X 239.959,Y -162.849,Z 164.969,A 145.837,B 90.000,C 0.000} C_DIS
LIN {X 239.613,Y -163.357,Z 165.075,A 145.716,B 90.000,C 0.000} C_DIS
LIN {X 238.653,Y -164.757,Z 165.113,A 145.380,B 90.000,C 0.000} C_DIS
LIN {X 238.303,Y -165.262,Z 165.220,A 145.259,B 90.000,C 0.000} C_DIS
LIN {X 237.331,Y -166.655,Z 165.258,A 144.923,B 90.000,C 0.000} C_DIS
LIN {X 236.988,Y -167.142,Z 165.364,A 144.806,B 90.000,C 0.000} C_DIS
LIN {X 236.068,Y -168.439,Z 165.403,A 144.491,B 90.000,C 0.000} C_DIS
LIN {X 235.695,Y -168.961,Z 165.509,A 144.365,B 90.000,C 0.000} C_DIS
LIN {X 234.331,Y -170.848,Z 165.528,A 143.905,B 90.000,C 0.000} C_DIS
LIN {X 233.862,Y -171.490,Z 164.763,A 143.748,B 90.000,C 0.000} C_DIS
LIN {X 233.719,Y -171.684,Z 164.661,A 143.700,B 90.000,C 0.000} C_DIS
LIN {X 233.642,Y -171.789,Z 164.682,A 143.674,B 90.000,C 0.000} C_DIS
LIN {X 233.572,Y -171.884,Z 164.784,A 143.651,B 90.000,C 0.000} C_DIS
LIN {X 233.390,Y -172.131,Z 164.827,A 143.590,B 90.000,C 0.000} C_DIS
LIN {X 233.315,Y -172.233,Z 164.929,A 143.565,B 90.000,C 0.000} C_DIS
LIN {X 233.133,Y -172.480,Z 164.971,A 143.505,B 90.000,C 0.000} C_DIS
LIN {X 233.057,Y -172.582,Z 165.073,A 143.480,B 90.000,C 0.000} C_DIS
LIN {X 232.874,Y -172.828,Z 165.116,A 143.419,B 90.000,C 0.000} C_DIS
LIN {X 232.836,Y -172.879,Z 165.167,A 143.406,B 90.000,C 0.000} C_DIS
LIN {X 232.811,Y -172.913,Z 165.218,A 143.398,B 90.000,C 0.000} C_DIS
LIN {X 232.689,Y -173.077,Z 165.260,A 143.358,B 90.000,C 0.000} C_DIS
LIN {X 232.664,Y -173.111,Z 165.311,A 143.349,B 90.000,C 0.000} C_DIS
LIN {X 232.626,Y -173.162,Z 165.362,A 143.337,B 90.000,C 0.000} C_DIS
LIN {X 232.443,Y -173.408,Z 165.405,A 143.276,B 90.000,C 0.000} C_DIS
LIN {X 232.367,Y -173.510,Z 165.507,A 143.251,B 90.000,C 0.000} C_DIS
LIN {X 232.184,Y -173.755,Z 165.549,A 143.191,B 90.000,C 0.000} C_DIS
LIN {X 232.107,Y -173.857,Z 165.651,A 143.165,B 90.000,C 0.000} C_DIS
LIN {X 231.923,Y -174.102,Z 165.694,A 143.105,B 90.000,C 0.000} C_DIS
LIN {X 231.885,Y -174.153,Z 165.745,A 143.092,B 90.000,C 0.000} C_DIS
LIN {X 231.860,Y -174.187,Z 165.796,A 143.084,B 90.000,C 0.000} C_DIS
LIN {X 231.737,Y -174.350,Z 165.838,A 143.044,B 90.000,C 0.000} C_DIS
LIN {X 231.712,Y -174.384,Z 165.889,A 143.035,B 90.000,C 0.000} C_DIS
LIN {X 231.673,Y -174.435,Z 165.940,A 143.023,B 90.000,C 0.000} C_DIS
LIN {X 231.489,Y -174.679,Z 165.983,A 142.962,B 90.000,C 0.000} C_DIS
LIN {X 231.412,Y -174.781,Z 166.085,A 142.937,B 90.000,C 0.000} C_DIS
LIN {X 231.227,Y -175.025,Z 166.127,A 142.876,B 90.000,C 0.000} C_DIS
